// TIA Portal V17 program export: 2 tag tables, 1 data types, 3 data blocks, 33 code blocks (in call order from the OBs), 23 instance data blocks

VAR_GLOBAL   // PLC tag table "Default tag table"
   System_Byte AT %MB1 : Byte;
   FirstScan AT %M1.0 : Bool;
   DiagStatusUpdate AT %M1.1 : Bool;
   Clock_Byte AT %MB0 : Byte;
   Clock_10Hz AT %M0.0 : Bool;
   Clock_5Hz AT %M0.1 : Bool;
   "Clock_2.5Hz" AT %M0.2 : Bool;
   Clock_2Hz AT %M0.3 : Bool;
   "Clock_1.25Hz" AT %M0.4 : Bool;
   Clock_1Hz AT %M0.5 : Bool;
   "Clock_0.625Hz" AT %M0.6 : Bool;
   "Clock_0.5Hz" AT %M0.7 : Bool;
   "System_Byte(1)" AT %MB1 : Byte;
   AlwaysTRUE AT %M1.2 : Bool;
   AlwaysFALSE AT %M1.3 : Bool;
   Tag_1 AT %Q0.0 : Bool;
   Tag_2 AT %Q0.7 : Bool;
END_VAR

VAR_GLOBAL   // PLC tag table "System_Tags"
   pulse_01s AT %M10.0 : Bool;
   pulse_05s AT %M10.1 : Bool;
   pulse_1s AT %M10.2 : Bool;
   pulse_5s AT %M10.3 : Bool;
   pulse_10s AT %M10.4 : Bool;
   pulse_30s AT %M10.5 : Bool;
   pulse_1m AT %M10.6 : Bool;
   pulse_5m AT %M10.7 : Bool;
   pulse_10m AT %M11.0 : Bool;
   pulse_1h AT %M11.2 : Bool;
   TRUE AT %M1.2 : Bool;
   FALSE AT %M1.3 : Bool;
   Hand_DI AT %M12.0 : Bool;
   Hand_DO AT %M12.1 : Bool;
   Hand_AI AT %M12.2 : Bool;
   Hand_AO AT %M12.3 : Bool;
   Hand_M AT %M12.4 : Bool;
   Hand_MD AT %M12.5 : Bool;
   Hand_MDA AT %M12.6 : Bool;
   Hand_V AT %M12.7 : Bool;
   Hand_VD2 AT %M13.0 : Bool;
   Hand_VDA AT %M13.1 : Bool;
   Hand_Any AT %M13.7 : Bool;
   Alm_AI AT %M14.0 : Bool;
   Alm_M AT %M14.1 : Bool;
   Alm_MD AT %M14.2 : Bool;
   Alm_MDA AT %M14.3 : Bool;
   Alm_V AT %M14.4 : Bool;
   Alm_VD2 AT %M14.5 : Bool;
   Alm_VDA AT %M14.6 : Bool;
   Alm_Logick AT %M14.7 : Bool;
   Alm_Any AT %M15.7 : Bool;
   All_Block AT %M2.0 : Bool;
   Reset_All AT %M3.0 : Bool;
   Local_Mode AT %M4.0 : Bool;
   Sim_All AT %M5.0 : Bool;
   AI_Val_1 AT %MB100 : Byte;
   AI_Val_2 AT %MB101 : Byte;
   AI_Value AT %MW100 : Word;
   AO_Val_1 AT %MB102 : Byte;
   AO_Val_2 AT %MB103 : Byte;
   AO_Value AT %MW102 : Word;
   Events AT %MW200 : Word;
   pulse_1_day AT %M11.3 : Bool;
   pulse_1_week AT %M11.4 : Bool;
   pulse_1_month AT %M11.5 : Bool;
   pulse_30m AT %M11.1 : Bool;
   pulse_s1 AT %M11.6 : Bool;
   pulse_s2 AT %M11.7 : Bool;
   Hand_Low AT %M13.5 : Bool;
   Hand_High AT %M13.6 : Bool;
   Reset_Hand AT %M3.1 : Bool;
   Events_pos AT %MW210 : Word;
   Alarms AT %MW202 : Word;
   Alarms_pos AT %MW212 : Word;
END_VAR

TYPE "CMD"
// stored: IsFailsafeCompliant false
   STRUCT
      Start_A : Bool;   // Автозапуск / Запуск в авторежиме
      Start_M : Bool;   // Ручной - вперёд / Запуск в ручном режиме
      Hand : Bool;   // 0 - авто, 1 - ручной / 0 - Авто, 1 - Ручной
      Local : Bool;   // Локальный
      Lock : Bool;   // Блокировать / Блокировка
      Service : Bool;   // Сервис
      Safety : Bool;   // Безопасность
      Force : Bool;   // Принудительный
      Alarm : Bool;   // Есть авария / Авария
      Reset : Bool;   // Сброс аварий
      Sim : Bool;   // Режим симуляции
      Vector { S7_SetPoint := 'True'} : Bool;   // Выбор направления
      ResetOpTime : Bool;   // Сброс счётчика наработки
      Ready : Bool := true;   // Разрешение дистанционного управления
      reserv : Bool;
   END_STRUCT;
END_TYPE

DATA_BLOCK "FE_DB"   // DB5
{ S7_Optimized_Access := 'FALSE' }
VERSION : 0.1
// stored: AutoNumber false, DBAccessibleFromOPCUA true, IsOnlyStoredInLoadMemory false, IsWriteProtectedInAS false
   VAR RETAIN
      FE : Array[0..1] of Struct   // Чтение - Input Register (04), Запись - Holding Register (06)
         Flow_Out : Real;   // Накопленный объем +
         Flow_In : Real;   // Накопленный объём -
         Flow : Real;   // Мгновенный расход
         TE_1 : Real;   // Температура канала 1, С
         TE_2 : Real;   // Температура канала 2, С
         PE : Real;   // Давление среды, кПа
         Use { S7_SetPoint := 'True'} : Bool;
         Link : Bool;
         NoRead : Bool;
         NoWrite : Bool;
         ID { S7_SetPoint := 'True'} : Int;
         ADDR { S7_SetPoint := 'True'} : UInt;
         "Name" { S7_SetPoint := 'True'} : String[10];
      END_STRUCT;
   END_VAR
BEGIN
   FE[0].Use := FALSE;
   FE[1].Use := TRUE;
   FE[0].ID := 0;
   FE[1].ID := 1;
   FE[0].ADDR := 0;
   FE[1].ADDR := 41;
   FE[0]."Name" := '';
   FE[1]."Name" := 'FE';
END_DATA_BLOCK

DATA_BLOCK "tGw_DB"   // DB3
{ S7_Optimized_Access := 'TRUE' }
VERSION : 0.1
// stored: AutoNumber true, DBAccessibleFromOPCUA true, IsOnlyStoredInLoadMemory false, IsRetainMemResEnabled false, IsWriteProtectedInAS false, MemoryReserve 100
   VAR RETAIN
      tGw : Array[0..1] of Struct   // Точка подключения к КП
         IP { S7_SetPoint := 'True'} : IP_V4;
         Port { S7_SetPoint := 'True'} : UInt;
      END_STRUCT;
      "Name" { S7_SetPoint := 'True'} : WString[10] := WSTRING#'1';
      ID { S7_SetPoint := 'True'} : Int := 0;
   END_VAR
BEGIN
   tGw[0].IP.ADDR[1] := 16#0A;
   tGw[0].IP.ADDR[2..3] := 16#01;
   tGw[0].IP.ADDR[4] := 16#9B;
   tGw[1].IP.ADDR[1] := 16#0A;
   tGw[1].IP.ADDR[2..3] := 16#01;
   tGw[1].IP.ADDR[4] := 16#C9;
   tGw[0..1].Port := 503;
END_DATA_BLOCK

DATA_BLOCK "Support_DB"   // DB1000
{ S7_Optimized_Access := 'TRUE' }
VERSION : 0.1
// stored: AutoNumber false, DBAccessibleFromOPCUA true, IsOnlyStoredInLoadMemory false, IsRetainMemResEnabled false, IsWriteProtectedInAS false, MemoryReserve 100
   VAR
      DTR_Clean : Bool;   // Очистка DTR
      DTR_1 : Int;   // Data Transfer 1
      DTR_2 : Int;   // Data Transfer 2
      DTR_3 : Int;   // Data Transfer 3
   END_VAR
   VAR RETAIN
      All_AIs { S7_SetPoint := 'True'} : Int := 399;   // Номер последнего DB аналоговых входов
      All_AOs { S7_SetPoint := 'True'} : Int := 499;   // Номер последнего DB аналоговых выходов
      All_DIs { S7_SetPoint := 'True'} : Int := 209;   // Номер последнего DB дискретных входов
      All_DOs { S7_SetPoint := 'True'} : Int := 219;   // Номер последнего DB дискретных выходов
      All_MDs { S7_SetPoint := 'True'} : Int := 599;   // Номер последнего DB двигателей без ЧП
      All_MDAs { S7_SetPoint := 'True'} : Int := 699;   // Номер последнего DB двигателей с ЧП
      All_VD2s { S7_SetPoint := 'True'} : Int := 799;   // Номер последнего DB заслонки
      All_VD2As { S7_SetPoint := 'True'} : Int := 899;   // Номер последнего DB заслонки с позиционированием
      All_PIDs { S7_SetPoint := 'True'} : Int := 999;   // Номер последнего DB для PID-регулятора
   END_VAR
BEGIN
END_DATA_BLOCK

ORGANIZATION_BLOCK "Main"   // OB1, LAD, ProgramCycle
TITLE = "Main Program Sweep (Cycle)"
{ S7_Optimized_Access := 'TRUE' }
VERSION : 0.1
// stored: AutoNumber true, IsIECCheckEnabled false, SetENOAutomatically false
   VAR_INPUT
      Initial_Call : Bool;   // Initial call of this OB
      Remanence : Bool;   // =True, if remanent data are available
   END_VAR
   VAR_TEMP   // added for the SCL form of the ladder/FBD networks
      _w1 : Bool;
   END_VAR
BEGIN

REGION Network 1
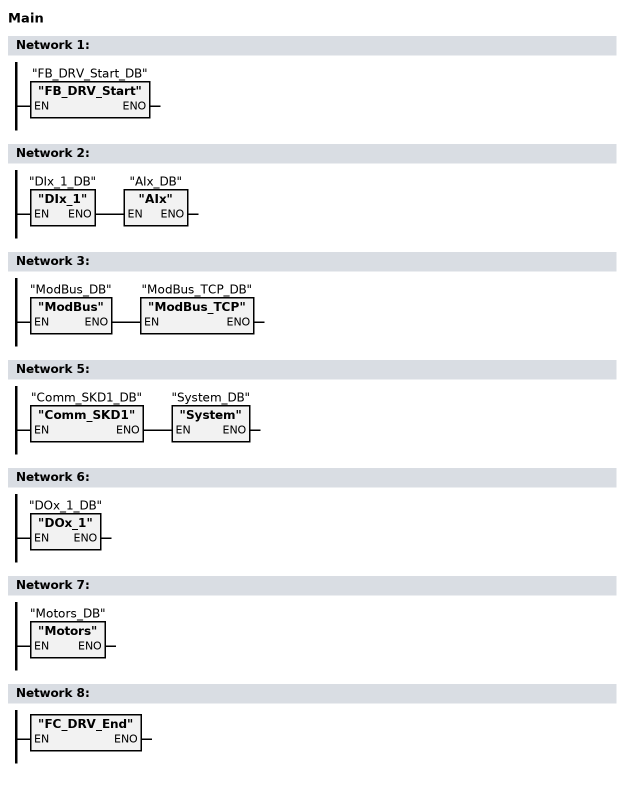
   RUNG wire#powerrail
      "FB_DRV_Start_DB"()
   END_RUNG
   // the same network as SCL:
   "FB_DRV_Start_DB"();   // "FB_DRV_Start"
END_REGION

REGION Network 2
   RUNG wire#powerrail
      "DIx_1_DB"()
      "AIx_DB"()
   END_RUNG
   // the same network as SCL:
   "DIx_1_DB"(ENO => #_w1);   // "DIx_1"
   IF #_w1 THEN
       "AIx_DB"();   // "AIx"
   END_IF;
END_REGION

REGION Network 3
   RUNG wire#powerrail
      "ModBus_DB"()
      "ModBus_TCP_DB"()
   END_RUNG
   // the same network as SCL:
   "ModBus_DB"(ENO => #_w1);   // "ModBus"
   IF #_w1 THEN
       "ModBus_TCP_DB"();   // "ModBus_TCP"
   END_IF;
END_REGION

REGION Network 5
   RUNG wire#powerrail
      "Comm_SKD1_DB"()
      "System_DB"()
   END_RUNG
   // the same network as SCL:
   "Comm_SKD1_DB"(ENO => #_w1);   // "Comm_SKD1"
   IF #_w1 THEN
       "System_DB"();   // "System"
   END_IF;
END_REGION

REGION Network 6
   RUNG wire#powerrail
      "DOx_1_DB"()
   END_RUNG
   // the same network as SCL:
   "DOx_1_DB"();   // "DOx_1"
END_REGION

REGION Network 7
   RUNG wire#powerrail
      "Motors_DB"()
   END_RUNG
   // the same network as SCL:
   "Motors_DB"();   // "Motors"
END_REGION

REGION Network 8
   RUNG wire#powerrail
      "FC_DRV_End"()
   END_RUNG
   // the same network as SCL:
   "FC_DRV_End"();
END_REGION
END_ORGANIZATION_BLOCK

FUNCTION_BLOCK "FB_DRV_Start"   // FB100, LAD
{ S7_Optimized_Access := 'TRUE' }
VERSION : 0.1
// stored: AutoNumber false, IsIECCheckEnabled false, IsRetainMemResEnabled false, MemoryReserve 100, SetENOAutomatically false, UDAEnableTagReadback false
   VAR
      last_01s : Int;
      last_05s : Int;
      last_1s : Int;
      last_5s : Int;
      last_10s : Int;
      last_30s : Int;
      last_1m : Int;
      last_5m : Int;
      last_10m : Int;
      last_30m : Int;
      last_1h : Int;
      last_1_day : Int;
      last_1_week : Int;
      last_1_month : Int;
      last_s1 : Int;
      last_s2 : Int;
      "1h_minutes" { S7_SetPoint := 'True'} : Int;
      "1_day_hour" { S7_SetPoint := 'True'} : Int;
      "1_day_minutes" { S7_SetPoint := 'True'} : Int;
      "1_week_weekday" { S7_SetPoint := 'True'} : Int := 1;
      "1_week_hour" { S7_SetPoint := 'True'} : Int;
      "1_week_minutes" { S7_SetPoint := 'True'} : Int;
      "1_month_date" { S7_SetPoint := 'True'} : Int := 1;
      "1_month_hour" { S7_SetPoint := 'True'} : Int;
      "1_month_minutes" { S7_SetPoint := 'True'} : Int;
      s1_hour : Int := 8;
      s1_minutes : Int;
      s2_hour : Int := 20;
      s2_minutes : Int;
      pos : Array[0..15] of Bool;
      Error : Word;
   END_VAR
   VAR_TEMP
      cnt_01s : Int;
      cnt_5s : Int;
      cnt_10s : Int;
      cnt_30s : Int;
      cnt_5m : Int;
      cnt_10m : Int;
      cnt_30m : Int;
   END_VAR
   VAR_TEMP   // added for the SCL form of the ladder/FBD networks
      _w1 : Bool;
      _w2 : Bool;
   END_VAR
BEGIN

REGION Network 1: Обработчик системного времени
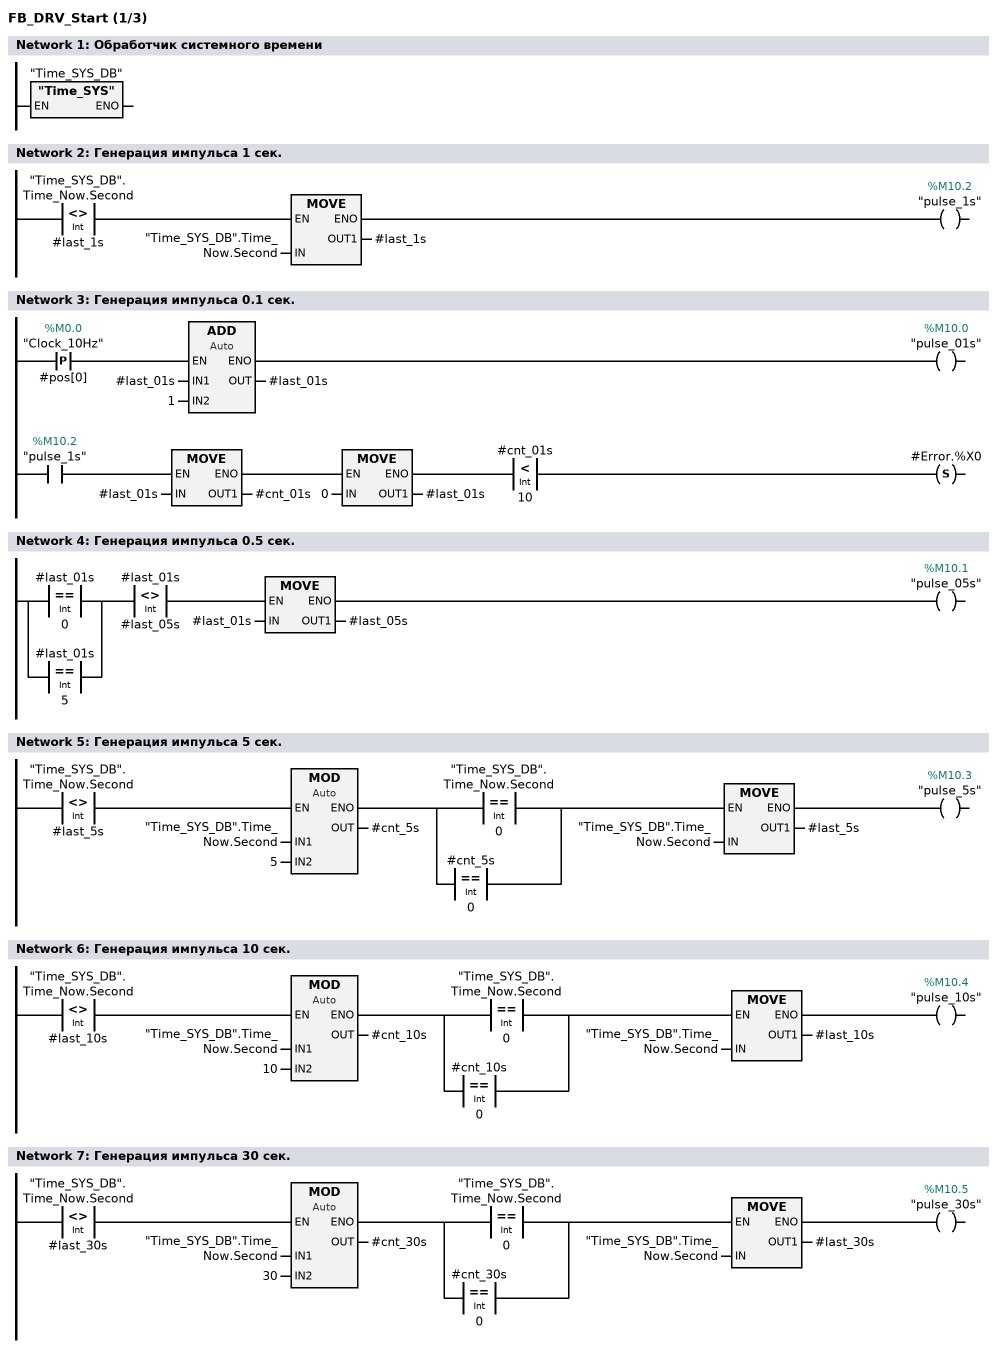
   RUNG wire#powerrail
      "Time_SYS_DB"()
   END_RUNG
   // the same network as SCL:
   "Time_SYS_DB"();   // "Time_SYS"
END_REGION

REGION Network 2: Генерация импульса 1 сек.
   RUNG wire#powerrail
      { S7_Templates := "SrcType := Int" } NE_Contact(in1 := "Time_SYS_DB".Time_Now.Second, in2 := #last_1s)
      Move(in := "Time_SYS_DB".Time_Now.Second, out1 => #last_1s)
      Coil( "pulse_1s" )
   END_RUNG
   // the same network as SCL:
   #_w1 := "Time_SYS_DB".Time_Now.Second <> #last_1s;
   IF #_w1 THEN #last_1s := "Time_SYS_DB".Time_Now.Second; END_IF;
   "pulse_1s" := #_w1;
END_REGION

REGION Network 3: Генерация импульса 0.1 сек.
   RUNG wire#powerrail
      P_Contact(operand := "Clock_10Hz", bit := #pos[0])
      Add(in1 := #last_01s, in2 := 1, out => #last_01s)
      Coil( "pulse_01s" )
   END_RUNG
   RUNG wire#powerrail
      Contact( "pulse_1s" )
      Move(in := #last_01s, out1 => #cnt_01s)
      Move(in := 0, out1 => #last_01s)
      { S7_Templates := "SrcType := Int" } LT_Contact(in1 := #cnt_01s, in2 := 10)
      S_Coil( #Error.%X0 )
   END_RUNG
   // the same network as SCL:
   #_w1 := "Clock_10Hz" AND NOT #pos[0];   // rising edge of "Clock_10Hz"
   #pos[0] := "Clock_10Hz";
   IF #_w1 THEN #last_01s := #last_01s + 1; END_IF;
   "pulse_01s" := #_w1;
   IF "pulse_1s" THEN
       #cnt_01s := #last_01s;
       #last_01s := 0;
   END_IF;
   IF "pulse_1s" AND (#cnt_01s < 10) THEN #Error.%X0 := TRUE; END_IF;
END_REGION

REGION Network 4: Генерация импульса 0.5 сек.
   RUNG wire#powerrail
      { S7_Templates := "SrcType := Int" } EQ_Contact(in1 := #last_01s, in2 := 0)
      wire#w1
      { S7_Templates := "SrcType := Int" } NE_Contact(in1 := #last_01s, in2 := #last_05s)
      Move(in := #last_01s, out1 => #last_05s)
      Coil( "pulse_05s" )
   END_RUNG
   RUNG wire#powerrail
      { S7_Templates := "SrcType := Int" } EQ_Contact(in1 := #last_01s, in2 := 5)
   END_RUNG wire#w1
   // the same network as SCL:
   #_w1 := ((#last_01s = 0) OR (#last_01s = 5)) AND (#last_01s <> #last_05s);
   IF #_w1 THEN #last_05s := #last_01s; END_IF;
   "pulse_05s" := #_w1;
END_REGION

REGION Network 5: Генерация импульса 5 сек.
   RUNG wire#powerrail
      { S7_Templates := "SrcType := Int" } NE_Contact(in1 := "Time_SYS_DB".Time_Now.Second, in2 := #last_5s)
      Mod(in1 := "Time_SYS_DB".Time_Now.Second, in2 := 5, out => #cnt_5s)
      wire#w1
      { S7_Templates := "SrcType := Int" } EQ_Contact(in1 := "Time_SYS_DB".Time_Now.Second, in2 := 0)
      wire#w2
      Move(in := "Time_SYS_DB".Time_Now.Second, out1 => #last_5s)
      Coil( "pulse_5s" )
   END_RUNG
   RUNG wire#w1
      { S7_Templates := "SrcType := Int" } EQ_Contact(in1 := #cnt_5s, in2 := 0)
   END_RUNG wire#w2
   // the same network as SCL:
   #_w1 := "Time_SYS_DB".Time_Now.Second <> #last_5s;
   IF #_w1 THEN #cnt_5s := "Time_SYS_DB".Time_Now.Second MOD 5; END_IF;
   #_w2 := #_w1 AND (("Time_SYS_DB".Time_Now.Second = 0) OR (#cnt_5s = 0));
   IF #_w2 THEN #last_5s := "Time_SYS_DB".Time_Now.Second; END_IF;
   "pulse_5s" := #_w2;
END_REGION

REGION Network 6: Генерация импульса 10 сек.
   RUNG wire#powerrail
      { S7_Templates := "SrcType := Int" } NE_Contact(in1 := "Time_SYS_DB".Time_Now.Second, in2 := #last_10s)
      Mod(in1 := "Time_SYS_DB".Time_Now.Second, in2 := 10, out => #cnt_10s)
      wire#w1
      { S7_Templates := "SrcType := Int" } EQ_Contact(in1 := "Time_SYS_DB".Time_Now.Second, in2 := 0)
      wire#w2
      Move(in := "Time_SYS_DB".Time_Now.Second, out1 => #last_10s)
      Coil( "pulse_10s" )
   END_RUNG
   RUNG wire#w1
      { S7_Templates := "SrcType := Int" } EQ_Contact(in1 := #cnt_10s, in2 := 0)
   END_RUNG wire#w2
   // the same network as SCL:
   #_w1 := "Time_SYS_DB".Time_Now.Second <> #last_10s;
   IF #_w1 THEN #cnt_10s := "Time_SYS_DB".Time_Now.Second MOD 10; END_IF;
   #_w2 := #_w1 AND (("Time_SYS_DB".Time_Now.Second = 0) OR (#cnt_10s = 0));
   IF #_w2 THEN #last_10s := "Time_SYS_DB".Time_Now.Second; END_IF;
   "pulse_10s" := #_w2;
END_REGION

REGION Network 7: Генерация импульса 30 сек.
   RUNG wire#powerrail
      { S7_Templates := "SrcType := Int" } NE_Contact(in1 := "Time_SYS_DB".Time_Now.Second, in2 := #last_30s)
      Mod(in1 := "Time_SYS_DB".Time_Now.Second, in2 := 30, out => #cnt_30s)
      wire#w1
      { S7_Templates := "SrcType := Int" } EQ_Contact(in1 := "Time_SYS_DB".Time_Now.Second, in2 := 0)
      wire#w2
      Move(in := "Time_SYS_DB".Time_Now.Second, out1 => #last_30s)
      Coil( "pulse_30s" )
   END_RUNG
   RUNG wire#w1
      { S7_Templates := "SrcType := Int" } EQ_Contact(in1 := #cnt_30s, in2 := 0)
   END_RUNG wire#w2
   // the same network as SCL:
   #_w1 := "Time_SYS_DB".Time_Now.Second <> #last_30s;
   IF #_w1 THEN #cnt_30s := "Time_SYS_DB".Time_Now.Second MOD 30; END_IF;
   #_w2 := #_w1 AND (("Time_SYS_DB".Time_Now.Second = 0) OR (#cnt_30s = 0));
   IF #_w2 THEN #last_30s := "Time_SYS_DB".Time_Now.Second; END_IF;
   "pulse_30s" := #_w2;
END_REGION

REGION Network 8: Генерация импульса 1 мин.
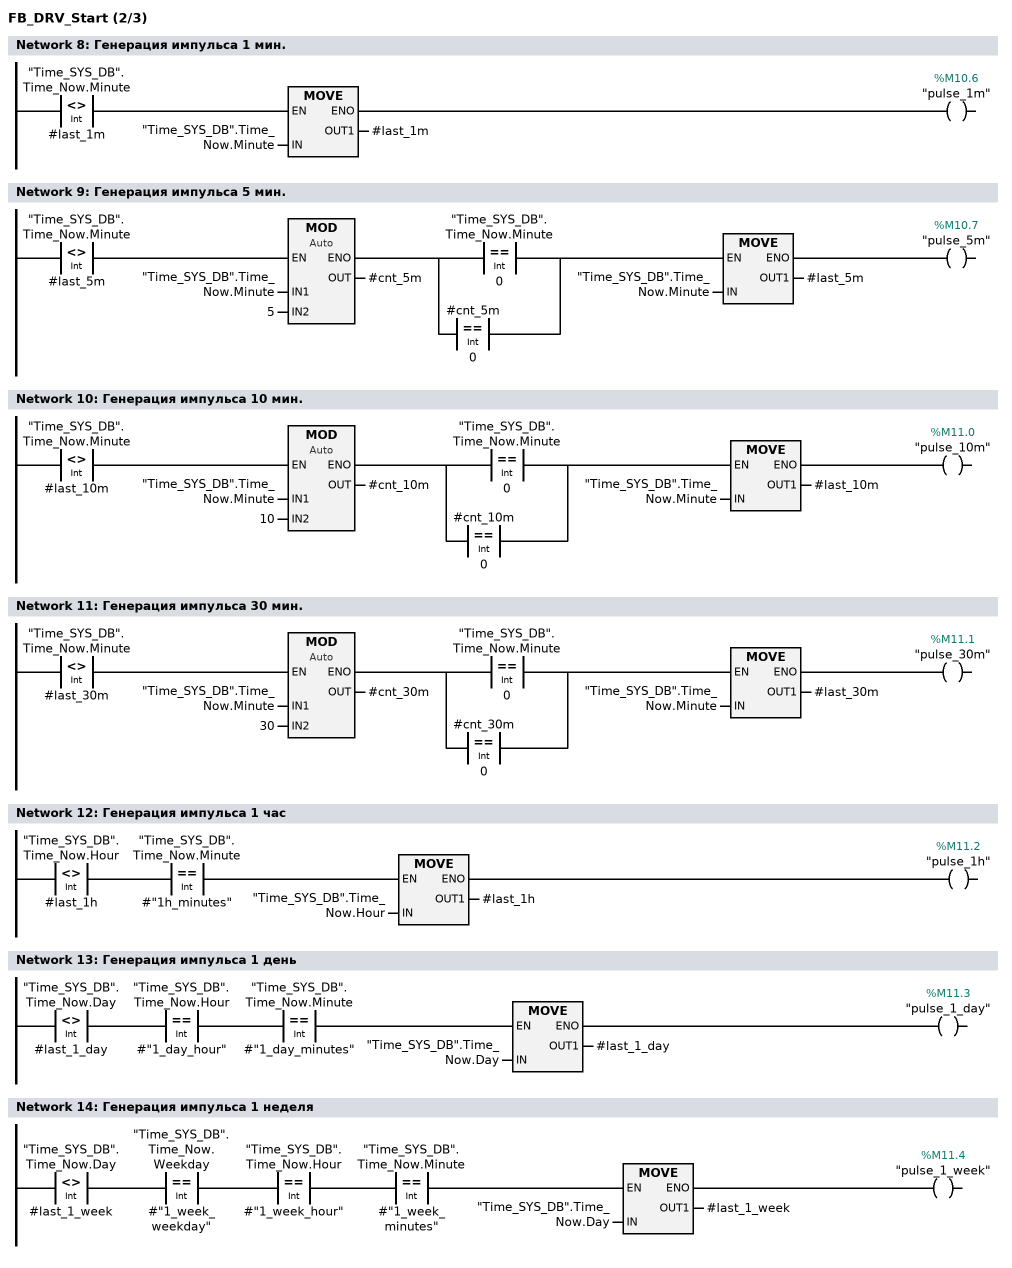
   RUNG wire#powerrail
      { S7_Templates := "SrcType := Int" } NE_Contact(in1 := "Time_SYS_DB".Time_Now.Minute, in2 := #last_1m)
      Move(in := "Time_SYS_DB".Time_Now.Minute, out1 => #last_1m)
      Coil( "pulse_1m" )
   END_RUNG
   // the same network as SCL:
   #_w1 := "Time_SYS_DB".Time_Now.Minute <> #last_1m;
   IF #_w1 THEN #last_1m := "Time_SYS_DB".Time_Now.Minute; END_IF;
   "pulse_1m" := #_w1;
END_REGION

REGION Network 9: Генерация импульса 5 мин.
   RUNG wire#powerrail
      { S7_Templates := "SrcType := Int" } NE_Contact(in1 := "Time_SYS_DB".Time_Now.Minute, in2 := #last_5m)
      Mod(in1 := "Time_SYS_DB".Time_Now.Minute, in2 := 5, out => #cnt_5m)
      wire#w1
      { S7_Templates := "SrcType := Int" } EQ_Contact(in1 := "Time_SYS_DB".Time_Now.Minute, in2 := 0)
      wire#w2
      Move(in := "Time_SYS_DB".Time_Now.Minute, out1 => #last_5m)
      Coil( "pulse_5m" )
   END_RUNG
   RUNG wire#w1
      { S7_Templates := "SrcType := Int" } EQ_Contact(in1 := #cnt_5m, in2 := 0)
   END_RUNG wire#w2
   // the same network as SCL:
   #_w1 := "Time_SYS_DB".Time_Now.Minute <> #last_5m;
   IF #_w1 THEN #cnt_5m := "Time_SYS_DB".Time_Now.Minute MOD 5; END_IF;
   #_w2 := #_w1 AND (("Time_SYS_DB".Time_Now.Minute = 0) OR (#cnt_5m = 0));
   IF #_w2 THEN #last_5m := "Time_SYS_DB".Time_Now.Minute; END_IF;
   "pulse_5m" := #_w2;
END_REGION

REGION Network 10: Генерация импульса 10 мин.
   RUNG wire#powerrail
      { S7_Templates := "SrcType := Int" } NE_Contact(in1 := "Time_SYS_DB".Time_Now.Minute, in2 := #last_10m)
      Mod(in1 := "Time_SYS_DB".Time_Now.Minute, in2 := 10, out => #cnt_10m)
      wire#w1
      { S7_Templates := "SrcType := Int" } EQ_Contact(in1 := "Time_SYS_DB".Time_Now.Minute, in2 := 0)
      wire#w2
      Move(in := "Time_SYS_DB".Time_Now.Minute, out1 => #last_10m)
      Coil( "pulse_10m" )
   END_RUNG
   RUNG wire#w1
      { S7_Templates := "SrcType := Int" } EQ_Contact(in1 := #cnt_10m, in2 := 0)
   END_RUNG wire#w2
   // the same network as SCL:
   #_w1 := "Time_SYS_DB".Time_Now.Minute <> #last_10m;
   IF #_w1 THEN #cnt_10m := "Time_SYS_DB".Time_Now.Minute MOD 10; END_IF;
   #_w2 := #_w1 AND (("Time_SYS_DB".Time_Now.Minute = 0) OR (#cnt_10m = 0));
   IF #_w2 THEN #last_10m := "Time_SYS_DB".Time_Now.Minute; END_IF;
   "pulse_10m" := #_w2;
END_REGION

REGION Network 11: Генерация импульса 30 мин.
   RUNG wire#powerrail
      { S7_Templates := "SrcType := Int" } NE_Contact(in1 := "Time_SYS_DB".Time_Now.Minute, in2 := #last_30m)
      Mod(in1 := "Time_SYS_DB".Time_Now.Minute, in2 := 30, out => #cnt_30m)
      wire#w1
      { S7_Templates := "SrcType := Int" } EQ_Contact(in1 := "Time_SYS_DB".Time_Now.Minute, in2 := 0)
      wire#w2
      Move(in := "Time_SYS_DB".Time_Now.Minute, out1 => #last_30m)
      Coil( "pulse_30m" )
   END_RUNG
   RUNG wire#w1
      { S7_Templates := "SrcType := Int" } EQ_Contact(in1 := #cnt_30m, in2 := 0)
   END_RUNG wire#w2
   // the same network as SCL:
   #_w1 := "Time_SYS_DB".Time_Now.Minute <> #last_30m;
   IF #_w1 THEN #cnt_30m := "Time_SYS_DB".Time_Now.Minute MOD 30; END_IF;
   #_w2 := #_w1 AND (("Time_SYS_DB".Time_Now.Minute = 0) OR (#cnt_30m = 0));
   IF #_w2 THEN #last_30m := "Time_SYS_DB".Time_Now.Minute; END_IF;
   "pulse_30m" := #_w2;
END_REGION

REGION Network 12: Генерация импульса 1 час
   RUNG wire#powerrail
      { S7_Templates := "SrcType := Int" } NE_Contact(in1 := "Time_SYS_DB".Time_Now.Hour, in2 := #last_1h)
      { S7_Templates := "SrcType := Int" } EQ_Contact(in1 := "Time_SYS_DB".Time_Now.Minute, in2 := #"1h_minutes")
      Move(in := "Time_SYS_DB".Time_Now.Hour, out1 => #last_1h)
      Coil( "pulse_1h" )
   END_RUNG
   // the same network as SCL:
   #_w1 := ("Time_SYS_DB".Time_Now.Hour <> #last_1h) AND ("Time_SYS_DB".Time_Now.Minute = #"1h_minutes");
   IF #_w1 THEN #last_1h := "Time_SYS_DB".Time_Now.Hour; END_IF;
   "pulse_1h" := #_w1;
END_REGION

REGION Network 13: Генерация импульса 1 день
   RUNG wire#powerrail
      { S7_Templates := "SrcType := Int" } NE_Contact(in1 := "Time_SYS_DB".Time_Now.Day, in2 := #last_1_day)
      { S7_Templates := "SrcType := Int" } EQ_Contact(in1 := "Time_SYS_DB".Time_Now.Hour, in2 := #"1_day_hour")
      { S7_Templates := "SrcType := Int" } EQ_Contact(in1 := "Time_SYS_DB".Time_Now.Minute, in2 := #"1_day_minutes")
      Move(in := "Time_SYS_DB".Time_Now.Day, out1 => #last_1_day)
      Coil( "pulse_1_day" )
   END_RUNG
   // the same network as SCL:
   #_w1 := ("Time_SYS_DB".Time_Now.Day <> #last_1_day) AND ("Time_SYS_DB".Time_Now.Hour = #"1_day_hour") AND ("Time_SYS_DB".Time_Now.Minute = #"1_day_minutes");
   IF #_w1 THEN #last_1_day := "Time_SYS_DB".Time_Now.Day; END_IF;
   "pulse_1_day" := #_w1;
END_REGION

REGION Network 14: Генерация импульса 1 неделя
   RUNG wire#powerrail
      { S7_Templates := "SrcType := Int" } NE_Contact(in1 := "Time_SYS_DB".Time_Now.Day, in2 := #last_1_week)
      { S7_Templates := "SrcType := Int" } EQ_Contact(in1 := "Time_SYS_DB".Time_Now.Weekday, in2 := #"1_week_weekday")
      { S7_Templates := "SrcType := Int" } EQ_Contact(in1 := "Time_SYS_DB".Time_Now.Hour, in2 := #"1_week_hour")
      { S7_Templates := "SrcType := Int" } EQ_Contact(in1 := "Time_SYS_DB".Time_Now.Minute, in2 := #"1_week_minutes")
      Move(in := "Time_SYS_DB".Time_Now.Day, out1 => #last_1_week)
      Coil( "pulse_1_week" )
   END_RUNG
   // the same network as SCL:
   #_w1 := ("Time_SYS_DB".Time_Now.Day <> #last_1_week) AND ("Time_SYS_DB".Time_Now.Weekday = #"1_week_weekday") AND ("Time_SYS_DB".Time_Now.Hour = #"1_week_hour") AND ("Time_SYS_DB".Time_Now.Minute = #"1_week_minutes");
   IF #_w1 THEN #last_1_week := "Time_SYS_DB".Time_Now.Day; END_IF;
   "pulse_1_week" := #_w1;
END_REGION

REGION Network 15: Генерация импульса 1 месяц
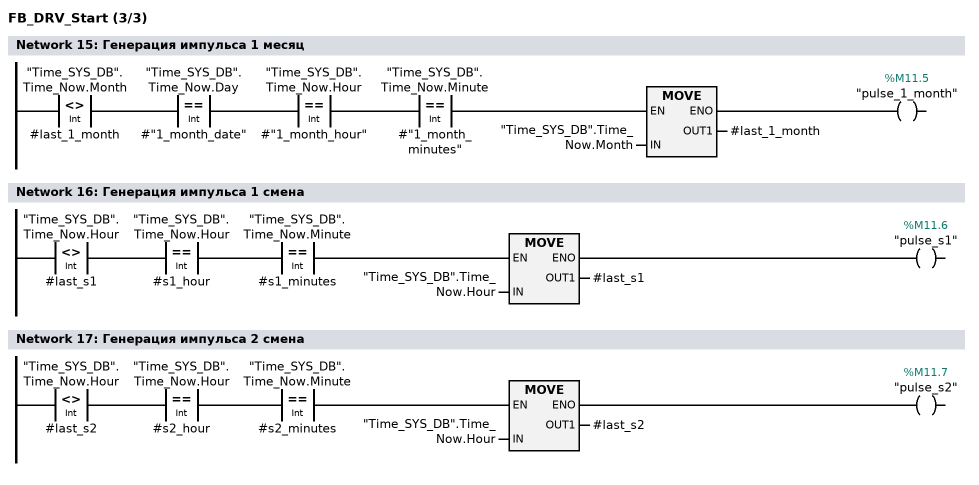
   RUNG wire#powerrail
      { S7_Templates := "SrcType := Int" } NE_Contact(in1 := "Time_SYS_DB".Time_Now.Month, in2 := #last_1_month)
      { S7_Templates := "SrcType := Int" } EQ_Contact(in1 := "Time_SYS_DB".Time_Now.Day, in2 := #"1_month_date")
      { S7_Templates := "SrcType := Int" } EQ_Contact(in1 := "Time_SYS_DB".Time_Now.Hour, in2 := #"1_month_hour")
      { S7_Templates := "SrcType := Int" } EQ_Contact(in1 := "Time_SYS_DB".Time_Now.Minute, in2 := #"1_month_minutes")
      Move(in := "Time_SYS_DB".Time_Now.Month, out1 => #last_1_month)
      Coil( "pulse_1_month" )
   END_RUNG
   // the same network as SCL:
   #_w1 := ("Time_SYS_DB".Time_Now.Month <> #last_1_month) AND ("Time_SYS_DB".Time_Now.Day = #"1_month_date") AND ("Time_SYS_DB".Time_Now.Hour = #"1_month_hour") AND ("Time_SYS_DB".Time_Now.Minute = #"1_month_minutes");
   IF #_w1 THEN #last_1_month := "Time_SYS_DB".Time_Now.Month; END_IF;
   "pulse_1_month" := #_w1;
END_REGION

REGION Network 16: Генерация импульса 1 смена
   RUNG wire#powerrail
      { S7_Templates := "SrcType := Int" } NE_Contact(in1 := "Time_SYS_DB".Time_Now.Hour, in2 := #last_s1)
      { S7_Templates := "SrcType := Int" } EQ_Contact(in1 := "Time_SYS_DB".Time_Now.Hour, in2 := #s1_hour)
      { S7_Templates := "SrcType := Int" } EQ_Contact(in1 := "Time_SYS_DB".Time_Now.Minute, in2 := #s1_minutes)
      Move(in := "Time_SYS_DB".Time_Now.Hour, out1 => #last_s1)
      Coil( "pulse_s1" )
   END_RUNG
   // the same network as SCL:
   #_w1 := ("Time_SYS_DB".Time_Now.Hour <> #last_s1) AND ("Time_SYS_DB".Time_Now.Hour = #s1_hour) AND ("Time_SYS_DB".Time_Now.Minute = #s1_minutes);
   IF #_w1 THEN #last_s1 := "Time_SYS_DB".Time_Now.Hour; END_IF;
   "pulse_s1" := #_w1;
END_REGION

REGION Network 17: Генерация импульса 2 смена
   RUNG wire#powerrail
      { S7_Templates := "SrcType := Int" } NE_Contact(in1 := "Time_SYS_DB".Time_Now.Hour, in2 := #last_s2)
      { S7_Templates := "SrcType := Int" } EQ_Contact(in1 := "Time_SYS_DB".Time_Now.Hour, in2 := #s2_hour)
      { S7_Templates := "SrcType := Int" } EQ_Contact(in1 := "Time_SYS_DB".Time_Now.Minute, in2 := #s2_minutes)
      Move(in := "Time_SYS_DB".Time_Now.Hour, out1 => #last_s2)
      Coil( "pulse_s2" )
   END_RUNG
   // the same network as SCL:
   #_w1 := ("Time_SYS_DB".Time_Now.Hour <> #last_s2) AND ("Time_SYS_DB".Time_Now.Hour = #s2_hour) AND ("Time_SYS_DB".Time_Now.Minute = #s2_minutes);
   IF #_w1 THEN #last_s2 := "Time_SYS_DB".Time_Now.Hour; END_IF;
   "pulse_s2" := #_w1;
END_REGION
END_FUNCTION_BLOCK

FUNCTION_BLOCK "Time_SYS"   // FB95, LAD
{ S7_Optimized_Access := 'FALSE' }
VERSION : 0.1
// stored: AutoNumber false, IsIECCheckEnabled false, SetENOAutomatically false, UDAEnableTagReadback false
   VAR DB_SPECIFIC
      Set_Time : Bool;   // Заданное время
      Time_Now : Struct   // Текущее время
         Year : Int;   // год
         Month : Int;   // месяц
         Day : Int;   // день месяца
         Weekday : Int;   // день недели (1 - воскресенье)
         Hour : Int;   // часы
         Minute : Int;   // минуты
         Second : Int;   // секунды
      END_STRUCT;
      Time_SP : Struct   // Текущее время
         Year : Int;   // год
         Month : Int;   // месяц
         Day : Int;   // день месяца
         Weekday : Int;   // день недели (1 - воскресенье)
         Hour : Int;   // часы
         Minute : Int;   // минуты
         Second : Int;   // секунды
      END_STRUCT;
      TimeZone { S7_SetPoint := 'True'} : TimeTransformationRule;   // Часовой пояс
      RD_SYS_Status : Int;   // Статус чтения времени
      WR_SYS_Status : Int;   // Статус записи времени
      RD_Time : DTL;   // Прочитанное сист. время
      SP_Time : DTL;   // Новое сист. время
   END_VAR
   VAR
      SET_TIMEZONE { S7_SetPoint := 'True'} : SET_TIMEZONE;   // Запись часового пояса
   END_VAR
   VAR DB_SPECIFIC
      Time_DTL : DTL;
   END_VAR
   // TimeZone.Bias := 180;   // Часовой пояс по GMT (смещение в минутах)
   // TimeZone.DaylightBias := 60;
   // TimeZone.DaylightStartMonth := 3;
   // TimeZone.DaylightStartWeek := 5;
   // TimeZone.DaylightStartWeekday := 7;
   // TimeZone.DaylightStartHour := 2;
   // TimeZone.DaylightStartMinute := 0;
   // TimeZone.StandardStartMonth := 10;
   // TimeZone.StandardStartWeek := 5;
   // TimeZone.StandardStartWeekday := 1;
   // TimeZone.StandardStartHour := 3;
   // TimeZone.StandardStartMinute := 0;
   // TimeZone.TimeZoneName := 'GMT+3';
   VAR_TEMP   // added for the SCL form of the ladder/FBD networks
      _w1 : Bool;
   END_VAR
BEGIN

REGION Network 1: Чтение системного времени
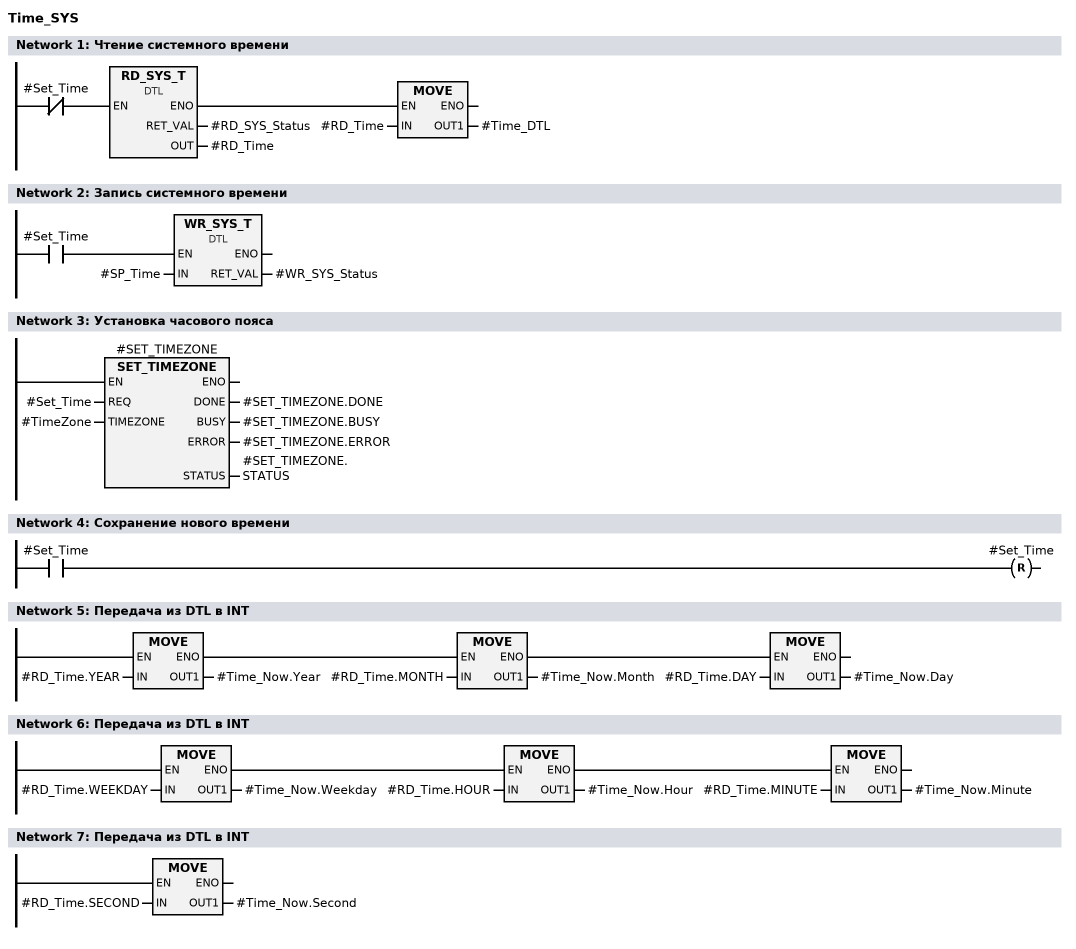
   RUNG wire#powerrail
      I_Contact( #Set_Time )
      { S7_Templates := "date_type := DTL" } RD_SYS_T(RET_VAL => #RD_SYS_Status, OUT => #RD_Time)
      Move(in := #RD_Time, out1 => #Time_DTL)
   END_RUNG
   // the same network as SCL:
   #RD_SYS_Status := RD_SYS_T(EN := NOT #Set_Time, OUT => #RD_Time, ENO => #_w1);
   IF #_w1 THEN #Time_DTL := #RD_Time; END_IF;
END_REGION

REGION Network 2: Запись системного времени
   RUNG wire#powerrail
      Contact( #Set_Time )
      { S7_Templates := "date_type := DTL" } WR_SYS_T(IN := #SP_Time, RET_VAL => #WR_SYS_Status)
   END_RUNG
   // the same network as SCL:
   IF #Set_Time THEN #WR_SYS_Status := WR_SYS_T(IN := #SP_Time); END_IF;
END_REGION

REGION Network 3: Установка часового пояса
   RUNG wire#powerrail
      #SET_TIMEZONE.SET_TIMEZONE(REQ := #Set_Time, TimeZone := #TimeZone, DONE => #SET_TIMEZONE.DONE, BUSY => #SET_TIMEZONE.BUSY, ERROR => #SET_TIMEZONE.ERROR, STATUS => #SET_TIMEZONE.STATUS)
   END_RUNG
   // the same network as SCL:
   #SET_TIMEZONE(REQ := #Set_Time,   // SET_TIMEZONE
                 TimeZone := #TimeZone,
                 DONE => #SET_TIMEZONE.DONE,
                 BUSY => #SET_TIMEZONE.BUSY,
                 ERROR => #SET_TIMEZONE.ERROR,
                 STATUS => #SET_TIMEZONE.STATUS);
END_REGION

REGION Network 4: Сохранение нового времени
   RUNG wire#powerrail
      Contact( #Set_Time )
      R_Coil( #Set_Time )
   END_RUNG
   // the same network as SCL:
   IF #Set_Time THEN #Set_Time := FALSE; END_IF;
END_REGION

REGION Network 5: Передача из DTL в INT
   RUNG wire#powerrail
      Move(in := #RD_Time.YEAR, out1 => #Time_Now.Year)
      Move(in := #RD_Time.MONTH, out1 => #Time_Now.Month)
      Move(in := #RD_Time.DAY, out1 => #Time_Now.Day)
   END_RUNG
   // the same network as SCL:
   #Time_Now.Year := #RD_Time.YEAR;
   #Time_Now.Month := #RD_Time.MONTH;
   #Time_Now.Day := #RD_Time.DAY;
END_REGION

REGION Network 6: Передача из DTL в INT
   RUNG wire#powerrail
      Move(in := #RD_Time.WEEKDAY, out1 => #Time_Now.Weekday)
      Move(in := #RD_Time.HOUR, out1 => #Time_Now.Hour)
      Move(in := #RD_Time.MINUTE, out1 => #Time_Now.Minute)
   END_RUNG
   // the same network as SCL:
   #Time_Now.Weekday := #RD_Time.WEEKDAY;
   #Time_Now.Hour := #RD_Time.HOUR;
   #Time_Now.Minute := #RD_Time.MINUTE;
END_REGION

REGION Network 7: Передача из DTL в INT
   RUNG wire#powerrail
      Move(in := #RD_Time.SECOND, out1 => #Time_Now.Second)
   END_RUNG
   // the same network as SCL:
   #Time_Now.Second := #RD_Time.SECOND;
END_REGION
END_FUNCTION_BLOCK

FUNCTION_BLOCK "DIx_1"   // FB200, LAD
{ S7_Optimized_Access := 'FALSE' }
VERSION : 0.1
// Input - входной сигнал контроллера
// pulse - частота фильтрации дребезга
// Signal - обработанный и отфильтрованный сигнал, используемый в дальнейшем
// stored: AutoNumber false, IsIECCheckEnabled false, SetENOAutomatically false, UDAEnableTagReadback false
   VAR
      AllBlock { S7_SetPoint := 'True'} : "DI_ex";   // Аварийный останов / 2.4 разрешение на работу
      "3FOk" { S7_SetPoint := 'True'} : "DI_ex";   // Питание в норме / 2.3 Нижний уровень
      Pump_Alarm { S7_SetPoint := 'True'} : "DI_ex";   // Авария насоса / Ротаметр 1
      Leak_KP { S7_SetPoint := 'True'} : "DI_ex";   // Затопление камеры КП2.7 / Ротаметр 2
      Level_Norm { S7_SetPoint := 'True'} : "DI_ex";   // Уровень в норме / Ротаметр 3
      "3Fok_1" { S7_SetPoint := 'True'} : "DI_ex";   // 3ф. сети Ввод 1 в норме / Датчик переливва
      "3Fok_2" { S7_SetPoint := 'True'} : "DI_ex";   // 3ф. сети Ввод 2 в норме / Датчик переливва
      "3Fok_sh" { S7_SetPoint := 'True'} : "DI_ex";   // 3ф. сети Ввод Шин в норме
      SHUSKV_Ok { S7_SetPoint := 'True'} : "DI_ex";   // Выключатель UC. Питание ШУСКВ в норме
      Leak_KP_res { S7_SetPoint := 'True'} : "DI_ex";
      Leak_KP_res_1 { S7_SetPoint := 'True'} : "DI_ex";
      signal_12 { S7_SetPoint := 'True'} : "DI_ex";
   END_VAR
   VAR DB_SPECIFIC
      Time_DTL { S7_SetPoint := 'True'} : DTL;
   END_VAR
   // AllBlock.ADDR_Bit := 3;
   // "3FOk".ADDR_Bit := 0;
   // Pump_Alarm.ADDR_Bit := 2;
   // Leak_KP.ADDR_Bit := 4;
   // Level_Norm.ADDR_Bit := 5;
   // "3Fok_1".ADDR_Bit := 6;
   // "3Fok_2".ADDR_Bit := 7;
   // "3Fok_sh".ADDR_Byte := 1;
   // "3Fok_sh".ADDR_Bit := 0;
   // SHUSKV_Ok.ADDR_Byte := 1;
   // SHUSKV_Ok.ADDR_Bit := 1;
   // Leak_KP_res.ADDR_Byte := 1;
   // Leak_KP_res.ADDR_Bit := 2;
   // Leak_KP_res_1.ADDR_Byte := 1;
   // Leak_KP_res_1.ADDR_Bit := 3;
   VAR_TEMP   // added for the SCL form of the ladder/FBD networks
      _w1 : Bool;
   END_VAR
BEGIN

REGION Network 1: AllBlock
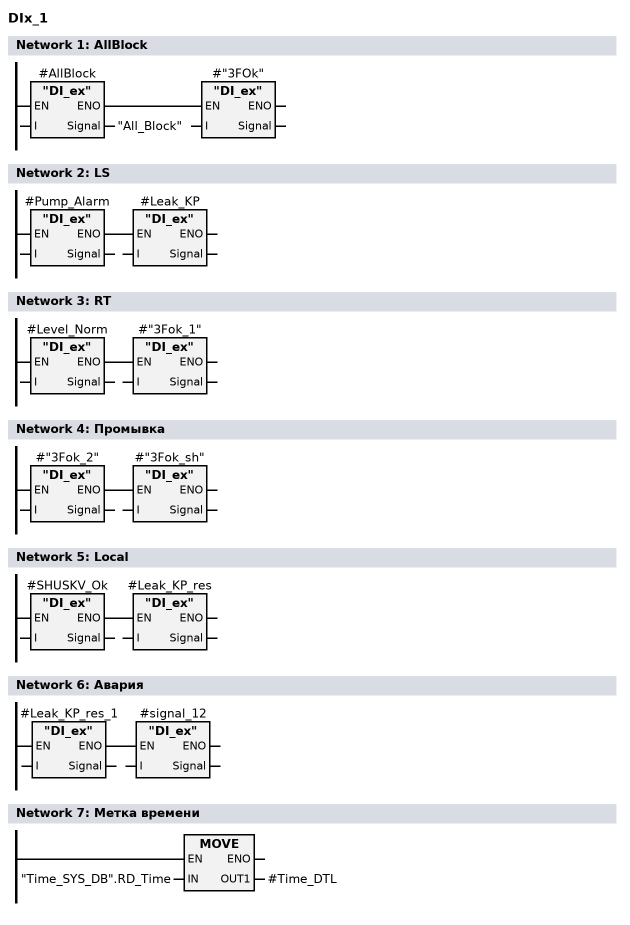
   RUNG wire#powerrail
      #AllBlock(I :=, Signal => "All_Block")
      #"3FOk"(I :=, Signal =>)
   END_RUNG
   // the same network as SCL:
   #AllBlock(Signal => "All_Block", ENO => #_w1);   // "DI_ex"
   IF #_w1 THEN
       #"3FOk"();   // "DI_ex"
   END_IF;
END_REGION

REGION Network 2: LS
   RUNG wire#powerrail
      #Pump_Alarm(I :=, Signal =>)
      #Leak_KP(I :=, Signal =>)
   END_RUNG
   // the same network as SCL:
   #Pump_Alarm(ENO => #_w1);   // "DI_ex"
   IF #_w1 THEN
       #Leak_KP();   // "DI_ex"
   END_IF;
END_REGION

REGION Network 3: RT
   RUNG wire#powerrail
      #Level_Norm(I :=, Signal =>)
      #"3Fok_1"(I :=, Signal =>)
   END_RUNG
   // the same network as SCL:
   #Level_Norm(ENO => #_w1);   // "DI_ex"
   IF #_w1 THEN
       #"3Fok_1"();   // "DI_ex"
   END_IF;
END_REGION

REGION Network 4: Промывка
   RUNG wire#powerrail
      #"3Fok_2"(I :=, Signal =>)
      #"3Fok_sh"(I :=, Signal =>)
   END_RUNG
   // the same network as SCL:
   #"3Fok_2"(ENO => #_w1);   // "DI_ex"
   IF #_w1 THEN
       #"3Fok_sh"();   // "DI_ex"
   END_IF;
END_REGION

REGION Network 5: Local
   RUNG wire#powerrail
      #SHUSKV_Ok(I :=, Signal =>)
      #Leak_KP_res(I :=, Signal =>)
   END_RUNG
   // the same network as SCL:
   #SHUSKV_Ok(ENO => #_w1);   // "DI_ex"
   IF #_w1 THEN
       #Leak_KP_res();   // "DI_ex"
   END_IF;
END_REGION

REGION Network 6: Авария
   RUNG wire#powerrail
      #Leak_KP_res_1(I :=, Signal =>)
      #signal_12(I :=, Signal =>)
   END_RUNG
   // the same network as SCL:
   #Leak_KP_res_1(ENO => #_w1);   // "DI_ex"
   IF #_w1 THEN
       #signal_12();   // "DI_ex"
   END_IF;
END_REGION

REGION Network 7: Метка времени
   RUNG wire#powerrail
      Move(in := "Time_SYS_DB".RD_Time, out1 => #Time_DTL)
   END_RUNG
   // the same network as SCL:
   #Time_DTL := "Time_SYS_DB".RD_Time;
END_REGION
END_FUNCTION_BLOCK

FUNCTION_BLOCK "DI_ex"   // FB101, LAD
{ S7_Optimized_Access := 'FALSE' }
VERSION : 0.1
// stored: AutoNumber false, IsIECCheckEnabled false, SetENOAutomatically false, UDAEnableTagReadback false
   VAR_INPUT
      I : Bool;   // Входной сигнал ПЛК
   END_VAR
   VAR_OUTPUT
      Signal : Bool;   // Результат обработки
   END_VAR
   VAR DB_SPECIFIC
      CMD : "CMD";   // Основные команды / Блок команд
      Use : Struct
         Inverse { S7_SetPoint := 'True'} : Bool;   // Инверсия входного сигнала
         Indirect { S7_SetPoint := 'True'} : Bool := true;   // Использование косвенной адресации
      END_STRUCT;
      ADDR_Byte { S7_SetPoint := 'True'} : Int;   // Адрес входа на контроллере (Байт)
      ADDR_Bit { S7_SetPoint := 'True'} : Int := 9;   // Адрес входа на контроллере (Бит)
   END_VAR
   VAR
      Filter_On { S7_SetPoint := 'True'} : "Time_S_b";   // Фильтр наличия сигнала
      Filter_Off { S7_SetPoint := 'True'} : "Time_S_b";   // Фильтр отсутствия сигнала
   END_VAR
   VAR_TEMP
      Data : Bool;
   END_VAR
   VAR_TEMP   // added for the SCL form of the ladder/FBD networks
      _w1 : Bool;
      _w2 : Bool;
   END_VAR
BEGIN

REGION Network 1: Устройство в ручном режиме
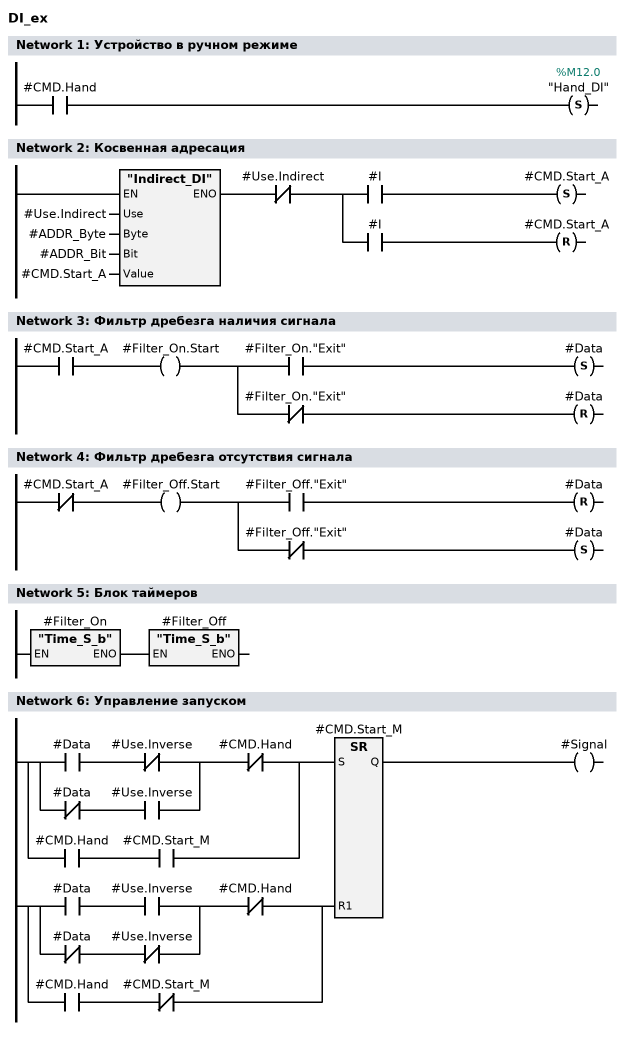
   RUNG wire#powerrail
      Contact( #CMD.Hand )
      S_Coil( "Hand_DI" )
   END_RUNG
   // the same network as SCL:
   IF #CMD.Hand THEN "Hand_DI" := TRUE; END_IF;
END_REGION

REGION Network 2: Косвенная адресация
   RUNG wire#powerrail
      "Indirect_DI"(Use := #Use.Indirect, "Byte" := #ADDR_Byte, Bit := #ADDR_Bit, Value := #CMD.Start_A)
      I_Contact( #Use.Indirect )
      wire#w1
      Contact( #I )
      S_Coil( #CMD.Start_A )
   END_RUNG
   RUNG wire#w1
      Contact( #I )
      R_Coil( #CMD.Start_A )
   END_RUNG
   // the same network as SCL:
   "Indirect_DI"(Use := #Use.Indirect,
                 "Byte" := #ADDR_Byte,
                 Bit := #ADDR_Bit,
                 Value := #CMD.Start_A,
                 ENO => #_w1);
   #_w2 := #_w1 AND NOT #Use.Indirect;
   IF #_w2 AND #I THEN
       #CMD.Start_A := TRUE;
       #CMD.Start_A := FALSE;
   END_IF;
END_REGION

REGION Network 3: Фильтр дребезга наличия сигнала
   RUNG wire#powerrail
      Contact( #CMD.Start_A )
      Coil( #Filter_On.Start )
      wire#w1
      Contact( #Filter_On."Exit" )
      S_Coil( #Data )
   END_RUNG
   RUNG wire#w1
      I_Contact( #Filter_On."Exit" )
      R_Coil( #Data )
   END_RUNG
   // the same network as SCL:
   #Filter_On.Start := #CMD.Start_A;
   IF #CMD.Start_A AND #Filter_On."Exit" THEN #Data := TRUE; END_IF;
   IF #CMD.Start_A AND NOT #Filter_On."Exit" THEN #Data := FALSE; END_IF;
END_REGION

REGION Network 4: Фильтр дребезга отсутствия сигнала
   RUNG wire#powerrail
      I_Contact( #CMD.Start_A )
      Coil( #Filter_Off.Start )
      wire#w1
      Contact( #Filter_Off."Exit" )
      R_Coil( #Data )
   END_RUNG
   RUNG wire#w1
      I_Contact( #Filter_Off."Exit" )
      S_Coil( #Data )
   END_RUNG
   // the same network as SCL:
   #Filter_Off.Start := NOT #CMD.Start_A;
   IF NOT #CMD.Start_A AND #Filter_Off."Exit" THEN #Data := FALSE; END_IF;
   IF NOT #CMD.Start_A AND NOT #Filter_Off."Exit" THEN #Data := TRUE; END_IF;
END_REGION

REGION Network 5: Блок таймеров
   RUNG wire#powerrail
      #Filter_On()
      #Filter_Off()
   END_RUNG
   // the same network as SCL:
   #Filter_On(ENO => #_w1);   // "Time_S_b"
   IF #_w1 THEN
       #Filter_Off();   // "Time_S_b"
   END_IF;
END_REGION

REGION Network 6: Управление запуском
   RUNG wire#powerrail
      Contact( #Data )
      I_Contact( #Use.Inverse )
      wire#w1
      I_Contact( #CMD.Hand )
      wire#w2
      S_SR(operand := #CMD.Start_M, r1 := wire#w4)
      Coil( #Signal )
   END_RUNG
   RUNG wire#powerrail
      I_Contact( #Data )
      Contact( #Use.Inverse )
   END_RUNG wire#w1
   RUNG wire#powerrail
      Contact( #CMD.Hand )
      Contact( #CMD.Start_M )
   END_RUNG wire#w2
   RUNG wire#powerrail
      Contact( #Data )
      Contact( #Use.Inverse )
      wire#w3
      I_Contact( #CMD.Hand )
   END_RUNG wire#w4
   RUNG wire#powerrail
      I_Contact( #Data )
      I_Contact( #Use.Inverse )
   END_RUNG wire#w3
   RUNG wire#powerrail
      Contact( #CMD.Hand )
      I_Contact( #CMD.Start_M )
   END_RUNG wire#w4
   // the same network as SCL:
   #_w1 := (((#Data AND #Use.Inverse) OR (NOT #Data AND NOT #Use.Inverse)) AND NOT #CMD.Hand) OR (#CMD.Hand AND NOT #CMD.Start_M);
   IF (((#Data AND NOT #Use.Inverse) OR (NOT #Data AND #Use.Inverse)) AND NOT #CMD.Hand) OR (#CMD.Hand AND #CMD.Start_M) THEN
       #CMD.Start_M := TRUE;   // SR flip-flop
   END_IF;
   IF #_w1 THEN #CMD.Start_M := FALSE; END_IF;
   #Signal := #CMD.Start_M;
END_REGION
END_FUNCTION_BLOCK

FUNCTION_BLOCK "Time_S_b"   // FB89, LAD
{ S7_Optimized_Access := 'FALSE' }
VERSION : 0.1
// stored: AutoNumber false, IsIECCheckEnabled false, SetENOAutomatically false, UDAEnableTagReadback false
   VAR DB_SPECIFIC
      SP { S7_SetPoint := 'True'} : Byte := 2;   // Уставка
      Now : Byte;   // Текущий счёт
      Start : Bool;   // Запуск
      "Exit" : Bool;   // Счёт завершён
      Pause : Bool;   // Пауза
      Reset : Bool;   // Сброс таймера
   END_VAR
   VAR_TEMP   // added for the SCL form of the ladder/FBD networks
      _w1 : Bool;
   END_VAR
BEGIN

REGION Network 1: Подсчёт времени
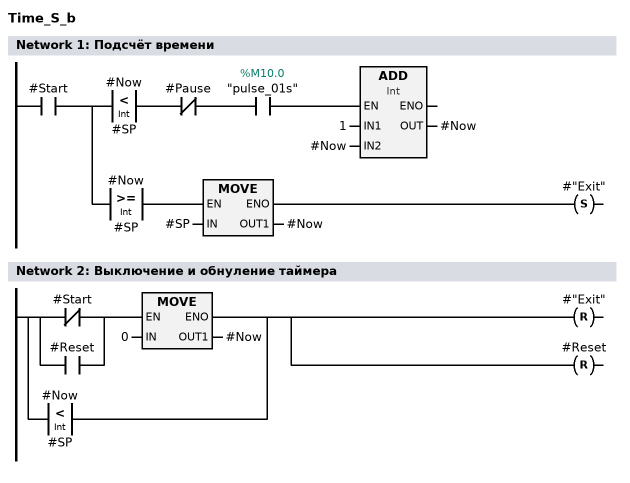
   RUNG wire#powerrail
      Contact( #Start )
      wire#w1
      { S7_Templates := "SrcType := Int" } LT_Contact(in1 := #Now, in2 := #SP)
      I_Contact( #Pause )
      Contact( "pulse_01s" )
      { S7_Templates := "SrcType := Int"; S7_GenerateENO := "TRUE" } Add(in1 := 1, in2 := #Now, out => #Now)
   END_RUNG
   RUNG wire#w1
      { S7_Templates := "SrcType := Int" } GE_Contact(in1 := #Now, in2 := #SP)
      { S7_GenerateENO := "TRUE" } Move(in := #SP, out1 => #Now)
      S_Coil( #"Exit" )
   END_RUNG
   // the same network as SCL:
   // ENO of a box is taken as its EN; it also drops when the box reports an error
   IF #Start AND (#Now < #SP) AND NOT #Pause AND "pulse_01s" THEN #Now := 1 + #Now; END_IF;
   #_w1 := #Start AND (#Now >= #SP);
   IF #_w1 THEN
       #Now := #SP;
       #"Exit" := TRUE;
   END_IF;
END_REGION

REGION Network 2: Выключение и обнуление таймера
   RUNG wire#powerrail
      I_Contact( #Start )
      wire#w1
      { S7_GenerateENO := "TRUE" } Move(in := 0, out1 => #Now)
      wire#w2
      R_Coil( #"Exit" )
   END_RUNG
   RUNG wire#powerrail
      Contact( #Reset )
   END_RUNG wire#w1
   RUNG wire#powerrail
      { S7_Templates := "SrcType := Int" } LT_Contact(in1 := #Now, in2 := #SP)
   END_RUNG wire#w2
   RUNG wire#w2
      R_Coil( #Reset )
   END_RUNG
   // the same network as SCL:
   // ENO of a box is taken as its EN; it also drops when the box reports an error
   #_w1 := NOT #Start OR #Reset;
   IF #_w1 THEN #Now := 0; END_IF;
   IF #_w1 OR (#Now < #SP) THEN
       #"Exit" := FALSE;
       #Reset := FALSE;
   END_IF;
END_REGION
END_FUNCTION_BLOCK

FUNCTION_BLOCK "AIx"   // FB220, LAD
{ S7_Optimized_Access := 'FALSE' }
VERSION : 0.1
// Signal - PIW код сигнала от датчика
// pulse - частота алгоритма фильтрации
// Result - результат обработки сигнала, формат Real
// stored: AutoNumber false, IsIECCheckEnabled false, SetENOAutomatically false, UDAEnableTagReadback false
   VAR DB_SPECIFIC
      Time_DTL { S7_SetPoint := 'True'} : DTL;
   END_VAR
   VAR_TEMP   // added for the SCL form of the ladder/FBD networks
      _w1 : Bool;
      _w2 : Bool;
   END_VAR
BEGIN

REGION Network 1: Датчик уровня
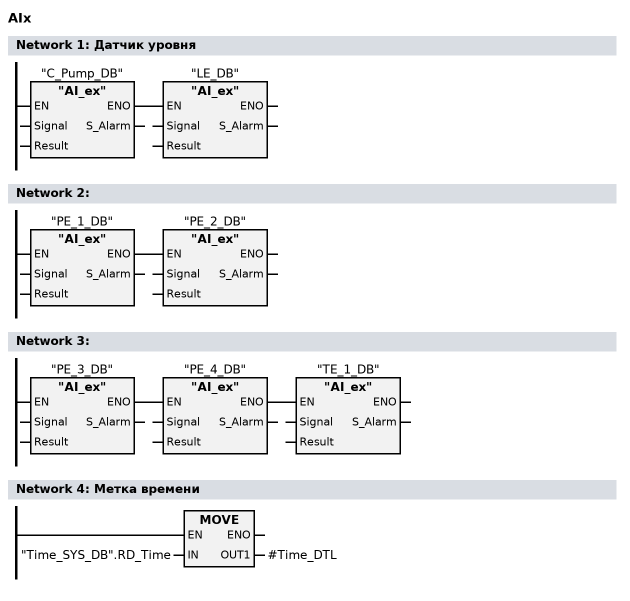
   RUNG wire#powerrail
      "C_Pump_DB"(Signal :=, Result :=, S_Alarm =>)
      "LE_DB"(Signal :=, Result :=, S_Alarm =>)
   END_RUNG
   // the same network as SCL:
   "C_Pump_DB"(ENO => #_w1);   // "AI_ex"
   IF #_w1 THEN
       "LE_DB"();   // "AI_ex"
   END_IF;
END_REGION

REGION Network 2
   RUNG wire#powerrail
      "PE_1_DB"(Signal :=, Result :=, S_Alarm =>)
      "PE_2_DB"(Signal :=, Result :=, S_Alarm =>)
   END_RUNG
   // the same network as SCL:
   "PE_1_DB"(ENO => #_w1);   // "AI_ex"
   IF #_w1 THEN
       "PE_2_DB"();   // "AI_ex"
   END_IF;
END_REGION

REGION Network 3
   RUNG wire#powerrail
      "PE_3_DB"(Signal :=, Result :=, S_Alarm =>)
      "PE_4_DB"(Signal :=, Result :=, S_Alarm =>)
      "TE_1_DB"(Signal :=, Result :=, S_Alarm =>)
   END_RUNG
   // the same network as SCL:
   "PE_3_DB"(ENO => #_w1);   // "AI_ex"
   "PE_4_DB"(EN := #_w1, ENO => #_w2);   // "AI_ex"
   IF #_w2 THEN
       "TE_1_DB"();   // "AI_ex"
   END_IF;
END_REGION

REGION Network 4: Метка времени
   RUNG wire#powerrail
      Move(in := "Time_SYS_DB".RD_Time, out1 => #Time_DTL)
   END_RUNG
   // the same network as SCL:
   #Time_DTL := "Time_SYS_DB".RD_Time;
END_REGION
END_FUNCTION_BLOCK

FUNCTION_BLOCK "AI_ex"   // FB103, LAD
{ S7_Optimized_Access := 'FALSE' }
VERSION : 0.1
// stored: AutoNumber false, IsIECCheckEnabled false, SetENOAutomatically false, UDAEnableTagReadback false
   VAR_OUTPUT
      S_Alarm : Bool;   // Внешний индикатор наличия аварии
   END_VAR
   VAR_IN_OUT
      Signal : Int;   // Входной сигнал контроллера
      Result : Real;   // Результат измерений
   END_VAR
   VAR DB_SPECIFIC
      CMD : "CMD";   // Основные команды / Блок команд
      Mode : Int;   // Режим работы
      Status : Int;   // Статус устройства
      Use : Struct   // Функционал
         RTD { S7_SetPoint := 'True'} : Bool;   // Режим RTD
         Filter { S7_SetPoint := 'True'} : Bool;   // Филтрация сигнала
         Inverse { S7_SetPoint := 'True'} : Bool;   // Инверсия сигнала
         Indirect { S7_SetPoint := 'True'} : Bool := true;   // Косвенная адресация
         Status { S7_SetPoint := 'True'} : Bool;   // Использовать подсветку
         Light { S7_SetPoint := 'True'} : Bool;   // Динамическая подсветка
         Lim_Low { S7_SetPoint := 'True'} : Bool;   // Отсечь низкие аварии
         Lim_High { S7_SetPoint := 'True'} : Bool;   // Отсечь высокие аварии
         Communication { S7_SetPoint := 'True'} : Bool;   // Передача в Value по сети
      END_STRUCT;
      VmA : Real;   // Реальный сигнал на входе ПЛК
      RTD_c { S7_SetPoint := 'True'} : Real := 10.0;   // Коэффициент RTD
      Calibration { S7_SetPoint := 'True'} : Real;   // Поправка
   END_VAR
   VAR
      Converter { S7_SetPoint := 'True'} : "Converter_LAD";   // Масштабирование сигнала
   END_VAR
   VAR DB_SPECIFIC
      SP : Struct   // Уставки аварий
         NC { S7_SetPoint := 'True'} : Real := -500.0;   // Сигнал при обрыве линии
         SC { S7_SetPoint := 'True'} : Real := 32000.0;   // Сигнал при КЗ/перегрузке
         HH { S7_SetPoint := 'True'} : Real := 90.0;   // Аварийно высокий сигнал
         H { S7_SetPoint := 'True'} : Real := 85.0;   // Высокий сигнал
         L { S7_SetPoint := 'True'} : Real := 15.0;   // Низкий сигнал
         LL { S7_SetPoint := 'True'} : Real := 10.0;   // Аварийно низкий сигнал
      END_STRUCT;
   END_VAR
   VAR
      Tx { S7_SetPoint := 'True'} : Array[0..5] of "Time_R";   // Блок таймеров
   END_VAR
   VAR DB_SPECIFIC
      Alarm : Struct   // Список аварий
         ST : Bool;   // Общая неисправность
         HH : Bool;   // сработала авария по аварийно высокму уровню
         H : Bool;   // сработало предупреждение по высокому уровню
         L : Bool;   // сработало предупреждение по низкому уровню
         LL : Bool;   // сработало предупрждение по аварийно низкому уровню
         NC : Bool;   // обрыв линии
         SC : Bool;   // короткое замыкание
      END_STRUCT;
      Alarms : Word;   // Слово аварий
      Events : Word;   // События датчика
      pos : Array[0..15] of Bool;   // Контроль фронтов событий
      Input_Type { S7_SetPoint := 'True'} : Int;   // Тип датчика, 0 - 4..20, 1 - 0..20, 2 - 0..10, 3 - 0..5, 4 - RTD
      CodeID { S7_SetPoint := 'True'} : Int;   // Код датчика для привязки в скаде
      "Type" { S7_SetPoint := 'True'} : Int;   // Тип датчика (единицы измерения)
      ADDR { S7_SetPoint := 'True'} : Int;   // Адрес входа на контроллере
      Filter_SP { S7_SetPoint := 'True'} : Int := 100;   // Ёмкость фильтра
      "Name" { S7_SetPoint := 'True'} : String[5];
   END_VAR
   VAR
      Filter_DB : "Filter";   // Фильтрация скачков сигнала
   END_VAR
   VAR DB_SPECIFIC
      Time_DTL { S7_SetPoint := 'True'} : DTL;
   END_VAR
   VAR_TEMP
      ev : Bool;   // Флаг событий
      Value : Real;   // Итоговый сигнал
      Signal_DI : DInt;   // Конвертация сигнала
      Signal_R : Real;   // Конвертация сигнала
      Type_Min : Real;
      Type_Max : Real;
   END_VAR
   VAR CONSTANT
      FALSE : Bool;
      TRUE : Bool := true;
   END_VAR
   // CMD.Start_A := true;
   // Converter.Max_In := 27648.0;
   // Converter.Max_Out := 100.0;
   VAR_TEMP   // added for the SCL form of the ladder/FBD networks
      _w1 : Bool;
      _w2 : Bool;
      _w3 : Bool;
      _w4 : Bool;
      _w5 : Bool;
      _w6 : Bool;
      _w7 : Bool;
      _w8 : Bool;
      _w9 : Bool;
      _w10 : Bool;
      _w11 : Bool;
      _w12 : Bool;
      _w13 : Bool;
      _w14 : Bool;
      _w15 : Bool;
      _w16 : Bool;
   END_VAR
BEGIN

REGION Network 1: Общий сброс
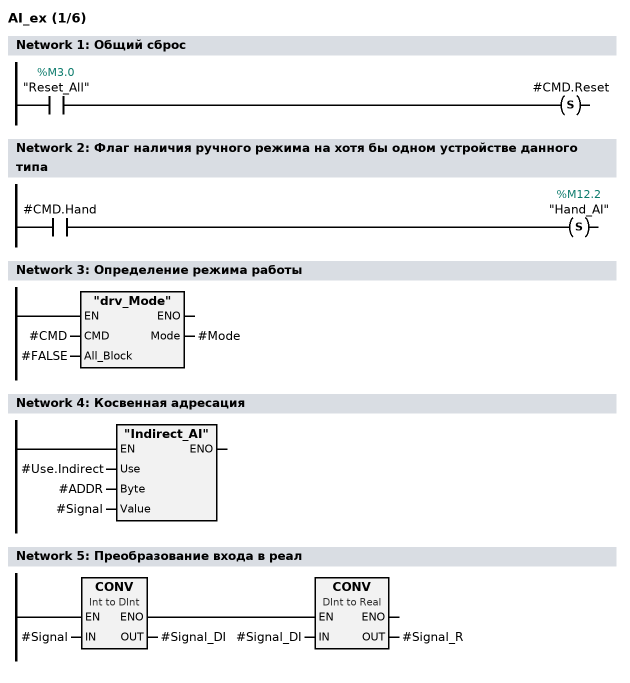
   RUNG wire#powerrail
      Contact( "Reset_All" )
      S_Coil( #CMD.Reset )
   END_RUNG
   // the same network as SCL:
   IF "Reset_All" THEN #CMD.Reset := TRUE; END_IF;
END_REGION

REGION Network 2: Флаг наличия ручного режима на хотя бы одном устройстве данного типа
   RUNG wire#powerrail
      Contact( #CMD.Hand )
      S_Coil( "Hand_AI" )
   END_RUNG
   // the same network as SCL:
   IF #CMD.Hand THEN "Hand_AI" := TRUE; END_IF;
END_REGION

REGION Network 3: Определение режима работы
   RUNG wire#powerrail
      "drv_Mode"(CMD := #CMD, All_Block := #FALSE, Mode => #Mode)
   END_RUNG
   // the same network as SCL:
   "drv_Mode"(CMD := #CMD, All_Block := #FALSE, Mode => #Mode);
END_REGION

REGION Network 4: Косвенная адресация
   RUNG wire#powerrail
      "Indirect_AI"(Use := #Use.Indirect, "Byte" := #ADDR, Value := #Signal)
   END_RUNG
   // the same network as SCL:
   "Indirect_AI"(Use := #Use.Indirect, "Byte" := #ADDR, Value := #Signal);
END_REGION

REGION Network 5: Преобразование входа в реал
   RUNG wire#powerrail
      { S7_Templates := "[SrcType := Int, DestType := DInt]"; S7_GenerateENO := "TRUE" } Convert(in := #Signal, out => #Signal_DI)
      { S7_Templates := "[SrcType := DInt, DestType := Real]"; S7_GenerateENO := "TRUE" } Convert(in := #Signal_DI, out => #Signal_R)
   END_RUNG
   // the same network as SCL:
   // ENO of a box is taken as its EN; it also drops when the box reports an error
   #Signal_DI := INT_TO_DINT(#Signal);
   #Signal_R := DINT_TO_REAL(#Signal_DI);
END_REGION

REGION Network 6: Преобразование кода в реальное значение входа
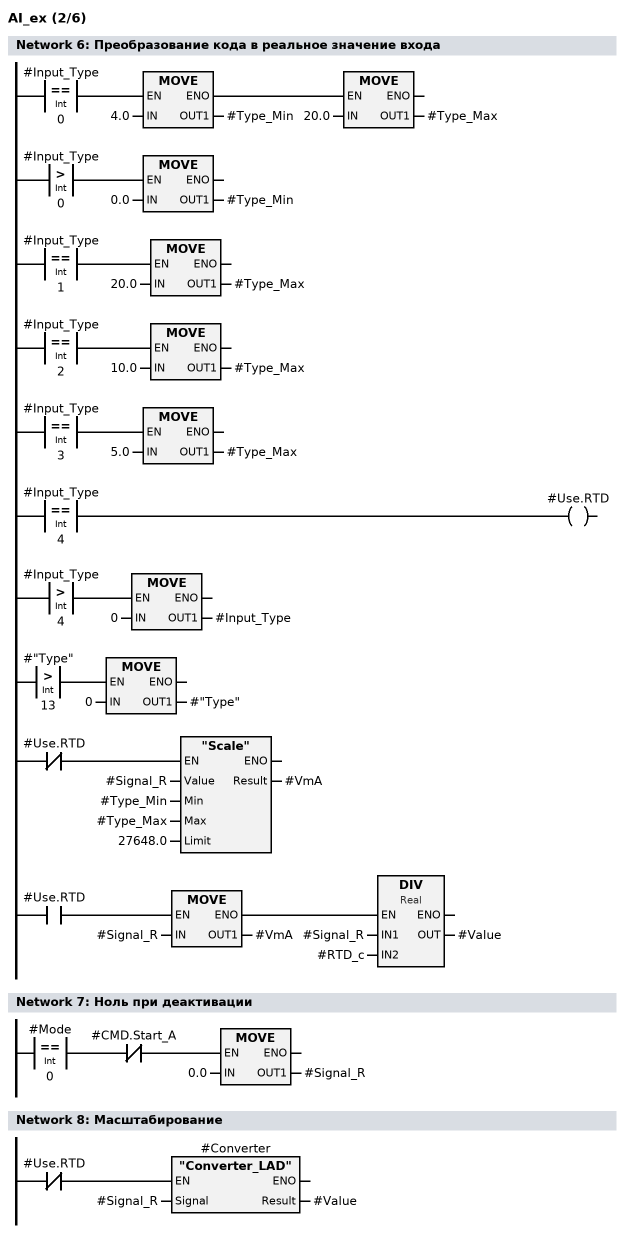
   RUNG wire#powerrail
      { S7_Templates := "SrcType := Int" } EQ_Contact(in1 := #Input_Type, in2 := 0)
      Move(in := 4.0, out1 => #Type_Min)
      Move(in := 20.0, out1 => #Type_Max)
   END_RUNG
   RUNG wire#powerrail
      { S7_Templates := "SrcType := Int" } GT_Contact(in1 := #Input_Type, in2 := 0)
      Move(in := 0.0, out1 => #Type_Min)
   END_RUNG
   RUNG wire#powerrail
      { S7_Templates := "SrcType := Int" } EQ_Contact(in1 := #Input_Type, in2 := 1)
      Move(in := 20.0, out1 => #Type_Max)
   END_RUNG
   RUNG wire#powerrail
      { S7_Templates := "SrcType := Int" } EQ_Contact(in1 := #Input_Type, in2 := 2)
      Move(in := 10.0, out1 => #Type_Max)
   END_RUNG
   RUNG wire#powerrail
      { S7_Templates := "SrcType := Int" } EQ_Contact(in1 := #Input_Type, in2 := 3)
      Move(in := 5.0, out1 => #Type_Max)
   END_RUNG
   RUNG wire#powerrail
      { S7_Templates := "SrcType := Int" } EQ_Contact(in1 := #Input_Type, in2 := 4)
      Coil( #Use.RTD )
   END_RUNG
   RUNG wire#powerrail
      { S7_Templates := "SrcType := Int" } GT_Contact(in1 := #Input_Type, in2 := 4)
      Move(in := 0, out1 => #Input_Type)
   END_RUNG
   RUNG wire#powerrail
      { S7_Templates := "SrcType := Int" } GT_Contact(in1 := #"Type", in2 := 13)
      Move(in := 0, out1 => #"Type")
   END_RUNG
   RUNG wire#powerrail
      I_Contact( #Use.RTD )
      "Scale"(Value := #Signal_R, Min := #Type_Min, Max := #Type_Max, Limit := 27648.0, Result => #VmA)
   END_RUNG
   RUNG wire#powerrail
      Contact( #Use.RTD )
      Move(in := #Signal_R, out1 => #VmA)
      { S7_Templates := "SrcType := Real"; S7_GenerateENO := "TRUE" } Div(in1 := #Signal_R, in2 := #RTD_c, out => #Value)
   END_RUNG
   // the same network as SCL:
   IF #Input_Type = 0 THEN
       #Type_Min := 4.0;
       #Type_Max := 20.0;
   END_IF;
   IF #Input_Type > 0 THEN #Type_Min := 0.0; END_IF;
   IF #Input_Type = 1 THEN #Type_Max := 20.0; END_IF;
   IF #Input_Type = 2 THEN #Type_Max := 10.0; END_IF;
   IF #Input_Type = 3 THEN #Type_Max := 5.0; END_IF;
   #Use.RTD := #Input_Type = 4;
   IF #Input_Type > 4 THEN #Input_Type := 0; END_IF;
   IF #"Type" > 13 THEN #"Type" := 0; END_IF;
   IF NOT #Use.RTD THEN
       "Scale"(Value := #Signal_R, Min := #Type_Min, Max := #Type_Max, Limit := 27648.0, Result => #VmA);
   END_IF;
   IF #Use.RTD THEN
       #VmA := #Signal_R;
       #Value := #Signal_R / #RTD_c;
   END_IF;
END_REGION

REGION Network 7: Ноль при деактивации
   RUNG wire#powerrail
      { S7_Templates := "SrcType := Int" } EQ_Contact(in1 := #Mode, in2 := 0)
      I_Contact( #CMD.Start_A )
      Move(in := 0.0, out1 => #Signal_R)
   END_RUNG
   // the same network as SCL:
   IF (#Mode = 0) AND NOT #CMD.Start_A THEN #Signal_R := 0.0; END_IF;
END_REGION

REGION Network 8: Масштабирование
   RUNG wire#powerrail
      I_Contact( #Use.RTD )
      #Converter(Signal := #Signal_R, Result => #Value)
   END_RUNG
   // the same network as SCL:
   IF NOT #Use.RTD THEN
       #Converter(Signal := #Signal_R, Result => #Value);   // "Converter_LAD"
   END_IF;
END_REGION

REGION Network 9: Вызов блока фильтрации
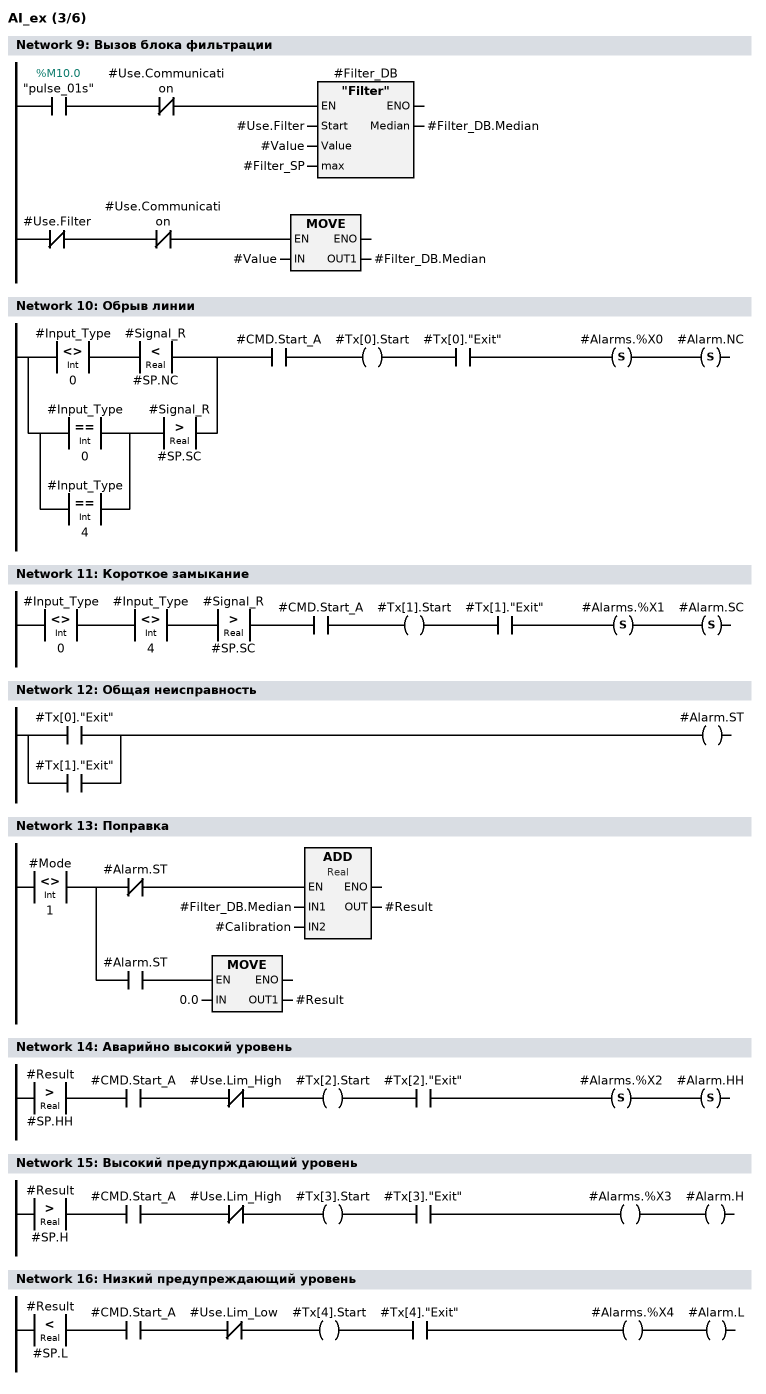
   RUNG wire#powerrail
      Contact( "pulse_01s" )
      I_Contact( #Use.Communication )
      #Filter_DB(Start := #Use.Filter, Value := #Value, max := #Filter_SP, Median => #Filter_DB.Median)
   END_RUNG
   RUNG wire#powerrail
      I_Contact( #Use.Filter )
      I_Contact( #Use.Communication )
      { S7_GenerateENO := "TRUE" } Move(in := #Value, out1 => #Filter_DB.Median)
   END_RUNG
   // the same network as SCL:
   IF "pulse_01s" AND NOT #Use.Communication THEN
       #Filter_DB(Start := #Use.Filter, Value := #Value, max := #Filter_SP, Median => #Filter_DB.Median);   // "Filter"
   END_IF;
   IF NOT #Use.Filter AND NOT #Use.Communication THEN #Filter_DB.Median := #Value; END_IF;
END_REGION

REGION Network 10: Обрыв линии
   RUNG wire#powerrail
      { S7_Templates := "SrcType := Int" } NE_Contact(in1 := #Input_Type, in2 := 0)
      { S7_Templates := "SrcType := Real" } LT_Contact(in1 := #Signal_R, in2 := #SP.NC)
      wire#w1
      Contact( #CMD.Start_A )
      Coil( #Tx[0].Start )
      Contact( #Tx[0]."Exit" )
      S_Coil( #Alarms.%X0 )
      S_Coil( #Alarm.NC )
   END_RUNG
   RUNG wire#powerrail
      { S7_Templates := "SrcType := Int" } EQ_Contact(in1 := #Input_Type, in2 := 0)
      wire#w2
      { S7_Templates := "SrcType := Real" } GT_Contact(in1 := #Signal_R, in2 := #SP.SC)
   END_RUNG wire#w1
   RUNG wire#powerrail
      { S7_Templates := "SrcType := Int" } EQ_Contact(in1 := #Input_Type, in2 := 4)
   END_RUNG wire#w2
   // the same network as SCL:
   #Tx[0].Start := (((#Input_Type <> 0) AND (#Signal_R < #SP.NC)) OR (((#Input_Type = 0) OR (#Input_Type = 4)) AND (#Signal_R > #SP.SC))) AND #CMD.Start_A;
   IF (((#Input_Type <> 0) AND (#Signal_R < #SP.NC)) OR (((#Input_Type = 0) OR (#Input_Type = 4)) AND (#Signal_R > #SP.SC))) AND #CMD.Start_A AND #Tx[0]."Exit" THEN
       #Alarms.%X0 := TRUE;
       #Alarm.NC := TRUE;
   END_IF;
END_REGION

REGION Network 11: Короткое замыкание
   RUNG wire#powerrail
      { S7_Templates := "SrcType := Int" } NE_Contact(in1 := #Input_Type, in2 := 0)
      { S7_Templates := "SrcType := Int" } NE_Contact(in1 := #Input_Type, in2 := 4)
      { S7_Templates := "SrcType := Real" } GT_Contact(in1 := #Signal_R, in2 := #SP.SC)
      Contact( #CMD.Start_A )
      Coil( #Tx[1].Start )
      Contact( #Tx[1]."Exit" )
      S_Coil( #Alarms.%X1 )
      S_Coil( #Alarm.SC )
   END_RUNG
   // the same network as SCL:
   #Tx[1].Start := (#Input_Type <> 0) AND (#Input_Type <> 4) AND (#Signal_R > #SP.SC) AND #CMD.Start_A;
   IF (#Input_Type <> 0) AND (#Input_Type <> 4) AND (#Signal_R > #SP.SC) AND #CMD.Start_A AND #Tx[1]."Exit" THEN
       #Alarms.%X1 := TRUE;
       #Alarm.SC := TRUE;
   END_IF;
END_REGION

REGION Network 12: Общая неисправность
   RUNG wire#powerrail
      Contact( #Tx[0]."Exit" )
      wire#w1
      Coil( #Alarm.ST )
   END_RUNG
   RUNG wire#powerrail
      Contact( #Tx[1]."Exit" )
   END_RUNG wire#w1
   // the same network as SCL:
   #Alarm.ST := #Tx[0]."Exit" OR #Tx[1]."Exit";
END_REGION

REGION Network 13: Поправка
   RUNG wire#powerrail
      { S7_Templates := "SrcType := Int" } NE_Contact(in1 := #Mode, in2 := 1)
      wire#w1
      I_Contact( #Alarm.ST )
      { S7_Templates := "SrcType := Real"; S7_GenerateENO := "TRUE" } Add(in1 := #Filter_DB.Median, in2 := #Calibration, out => #Result)
   END_RUNG
   RUNG wire#w1
      Contact( #Alarm.ST )
      Move(in := 0.0, out1 => #Result)
   END_RUNG
   // the same network as SCL:
   #_w1 := #Mode <> 1;
   IF #_w1 AND NOT #Alarm.ST THEN #Result := #Filter_DB.Median + #Calibration; END_IF;
   IF #_w1 AND #Alarm.ST THEN #Result := 0.0; END_IF;
END_REGION

REGION Network 14: Аварийно высокий уровень
   RUNG wire#powerrail
      { S7_Templates := "SrcType := Real" } GT_Contact(in1 := #Result, in2 := #SP.HH)
      Contact( #CMD.Start_A )
      I_Contact( #Use.Lim_High )
      Coil( #Tx[2].Start )
      Contact( #Tx[2]."Exit" )
      S_Coil( #Alarms.%X2 )
      S_Coil( #Alarm.HH )
   END_RUNG
   // the same network as SCL:
   #Tx[2].Start := (#Result > #SP.HH) AND #CMD.Start_A AND NOT #Use.Lim_High;
   IF (#Result > #SP.HH) AND #CMD.Start_A AND NOT #Use.Lim_High AND #Tx[2]."Exit" THEN
       #Alarms.%X2 := TRUE;
       #Alarm.HH := TRUE;
   END_IF;
END_REGION

REGION Network 15: Высокий предупрждающий уровень
   RUNG wire#powerrail
      { S7_Templates := "SrcType := Real" } GT_Contact(in1 := #Result, in2 := #SP.H)
      Contact( #CMD.Start_A )
      I_Contact( #Use.Lim_High )
      Coil( #Tx[3].Start )
      Contact( #Tx[3]."Exit" )
      Coil( #Alarms.%X3 )
      Coil( #Alarm.H )
   END_RUNG
   // the same network as SCL:
   #Tx[3].Start := (#Result > #SP.H) AND #CMD.Start_A AND NOT #Use.Lim_High;
   #Alarms.%X3 := (#Result > #SP.H) AND #CMD.Start_A AND NOT #Use.Lim_High AND #Tx[3]."Exit";
   #Alarm.H := #Alarms.%X3;
END_REGION

REGION Network 16: Низкий предупреждающий уровень
   RUNG wire#powerrail
      { S7_Templates := "SrcType := Real" } LT_Contact(in1 := #Result, in2 := #SP.L)
      Contact( #CMD.Start_A )
      I_Contact( #Use.Lim_Low )
      Coil( #Tx[4].Start )
      Contact( #Tx[4]."Exit" )
      Coil( #Alarms.%X4 )
      Coil( #Alarm.L )
   END_RUNG
   // the same network as SCL:
   #Tx[4].Start := (#Result < #SP.L) AND #CMD.Start_A AND NOT #Use.Lim_Low;
   #Alarms.%X4 := (#Result < #SP.L) AND #CMD.Start_A AND NOT #Use.Lim_Low AND #Tx[4]."Exit";
   #Alarm.L := #Alarms.%X4;
END_REGION

REGION Network 17: Аварийно высокий уровень
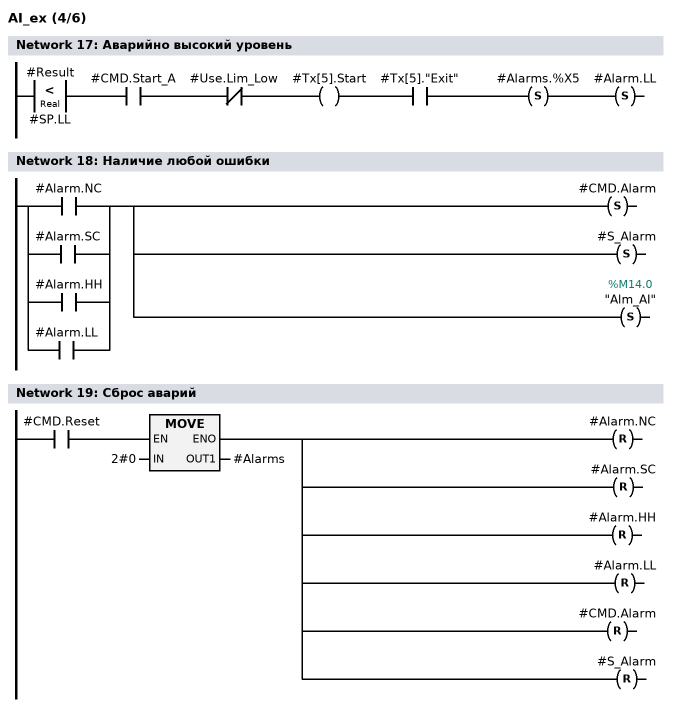
   RUNG wire#powerrail
      { S7_Templates := "SrcType := Real" } LT_Contact(in1 := #Result, in2 := #SP.LL)
      Contact( #CMD.Start_A )
      I_Contact( #Use.Lim_Low )
      Coil( #Tx[5].Start )
      Contact( #Tx[5]."Exit" )
      S_Coil( #Alarms.%X5 )
      S_Coil( #Alarm.LL )
   END_RUNG
   // the same network as SCL:
   #Tx[5].Start := (#Result < #SP.LL) AND #CMD.Start_A AND NOT #Use.Lim_Low;
   IF (#Result < #SP.LL) AND #CMD.Start_A AND NOT #Use.Lim_Low AND #Tx[5]."Exit" THEN
       #Alarms.%X5 := TRUE;
       #Alarm.LL := TRUE;
   END_IF;
END_REGION

REGION Network 18: Наличие любой ошибки
   RUNG wire#powerrail
      Contact( #Alarm.NC )
      wire#w1
      S_Coil( #CMD.Alarm )
   END_RUNG
   RUNG wire#powerrail
      Contact( #Alarm.SC )
   END_RUNG wire#w1
   RUNG wire#powerrail
      Contact( #Alarm.HH )
   END_RUNG wire#w1
   RUNG wire#powerrail
      Contact( #Alarm.LL )
   END_RUNG wire#w1
   RUNG wire#w1
      S_Coil( #S_Alarm )
   END_RUNG
   RUNG wire#w1
      S_Coil( "Alm_AI" )
   END_RUNG
   // the same network as SCL:
   IF #Alarm.NC OR #Alarm.SC OR #Alarm.HH OR #Alarm.LL THEN
       #CMD.Alarm := TRUE;
       #S_Alarm := TRUE;
       "Alm_AI" := TRUE;
   END_IF;
END_REGION

REGION Network 19: Сброс аварий
   RUNG wire#powerrail
      Contact( #CMD.Reset )
      Move(in := 2#0, out1 => #Alarms)
      wire#w1
      R_Coil( #Alarm.NC )
   END_RUNG
   RUNG wire#w1
      R_Coil( #Alarm.SC )
   END_RUNG
   RUNG wire#w1
      R_Coil( #Alarm.HH )
   END_RUNG
   RUNG wire#w1
      R_Coil( #Alarm.LL )
   END_RUNG
   RUNG wire#w1
      R_Coil( #CMD.Alarm )
   END_RUNG
   RUNG wire#w1
      R_Coil( #S_Alarm )
   END_RUNG
   // the same network as SCL:
   IF #CMD.Reset THEN
       #Alarms := 2#0;
       #Alarm.NC := FALSE;
       #Alarm.SC := FALSE;
       #Alarm.HH := FALSE;
       #Alarm.LL := FALSE;
       #CMD.Alarm := FALSE;
       #S_Alarm := FALSE;
   END_IF;
END_REGION

REGION Network 20: События датчика
   // 0 - датчик активирован
   // 1 - датчик деактивирован
   // 2 - датчик в ручном режиме
   // 3 - датчик в автоматическом режиме
   // 4 - сигнал ниже нижнего предупреждающего
   // 5 - сигнал в норме
   // 6 - сигнал выше верхнего предупреждающего
   // 7 - сигнал в норме
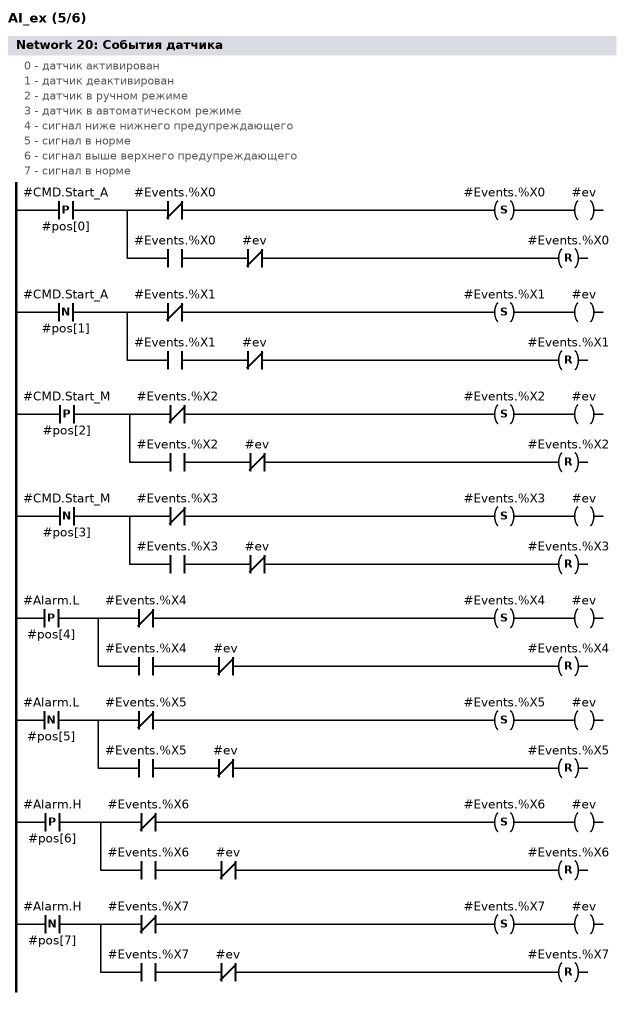
   RUNG wire#powerrail
      P_Contact(operand := #CMD.Start_A, bit := #pos[0])
      wire#w1
      I_Contact( #Events.%X0 )
      S_Coil( #Events.%X0 )
      Coil( #ev )
   END_RUNG
   RUNG wire#w1
      Contact( #Events.%X0 )
      I_Contact( #ev )
      R_Coil( #Events.%X0 )
   END_RUNG
   RUNG wire#powerrail
      N_Contact(operand := #CMD.Start_A, bit := #pos[1])
      wire#w2
      I_Contact( #Events.%X1 )
      S_Coil( #Events.%X1 )
      Coil( #ev )
   END_RUNG
   RUNG wire#w2
      Contact( #Events.%X1 )
      I_Contact( #ev )
      R_Coil( #Events.%X1 )
   END_RUNG
   RUNG wire#powerrail
      P_Contact(operand := #CMD.Start_M, bit := #pos[2])
      wire#w3
      I_Contact( #Events.%X2 )
      S_Coil( #Events.%X2 )
      Coil( #ev )
   END_RUNG
   RUNG wire#w3
      Contact( #Events.%X2 )
      I_Contact( #ev )
      R_Coil( #Events.%X2 )
   END_RUNG
   RUNG wire#powerrail
      N_Contact(operand := #CMD.Start_M, bit := #pos[3])
      wire#w4
      I_Contact( #Events.%X3 )
      S_Coil( #Events.%X3 )
      Coil( #ev )
   END_RUNG
   RUNG wire#w4
      Contact( #Events.%X3 )
      I_Contact( #ev )
      R_Coil( #Events.%X3 )
   END_RUNG
   RUNG wire#powerrail
      P_Contact(operand := #Alarm.L, bit := #pos[4])
      wire#w5
      I_Contact( #Events.%X4 )
      S_Coil( #Events.%X4 )
      Coil( #ev )
   END_RUNG
   RUNG wire#w5
      Contact( #Events.%X4 )
      I_Contact( #ev )
      R_Coil( #Events.%X4 )
   END_RUNG
   RUNG wire#powerrail
      N_Contact(operand := #Alarm.L, bit := #pos[5])
      wire#w6
      I_Contact( #Events.%X5 )
      S_Coil( #Events.%X5 )
      Coil( #ev )
   END_RUNG
   RUNG wire#w6
      Contact( #Events.%X5 )
      I_Contact( #ev )
      R_Coil( #Events.%X5 )
   END_RUNG
   RUNG wire#powerrail
      P_Contact(operand := #Alarm.H, bit := #pos[6])
      wire#w7
      I_Contact( #Events.%X6 )
      S_Coil( #Events.%X6 )
      Coil( #ev )
   END_RUNG
   RUNG wire#w7
      Contact( #Events.%X6 )
      I_Contact( #ev )
      R_Coil( #Events.%X6 )
   END_RUNG
   RUNG wire#powerrail
      N_Contact(operand := #Alarm.H, bit := #pos[7])
      wire#w8
      I_Contact( #Events.%X7 )
      S_Coil( #Events.%X7 )
      Coil( #ev )
   END_RUNG
   RUNG wire#w8
      Contact( #Events.%X7 )
      I_Contact( #ev )
      R_Coil( #Events.%X7 )
   END_RUNG
   // the same network as SCL:
   #_w1 := #CMD.Start_A AND NOT #pos[0];   // rising edge of #CMD.Start_A
   #pos[0] := #CMD.Start_A;
   #_w2 := #_w1 AND NOT #Events.%X0;
   IF #_w2 THEN #Events.%X0 := TRUE; END_IF;
   #ev := #_w2;
   IF #_w1 AND #Events.%X0 AND NOT #ev THEN #Events.%X0 := FALSE; END_IF;
   #_w3 := NOT #CMD.Start_A AND #pos[1];   // falling edge of #CMD.Start_A
   #pos[1] := #CMD.Start_A;
   #_w4 := #_w3 AND NOT #Events.%X1;
   IF #_w4 THEN #Events.%X1 := TRUE; END_IF;
   #ev := #_w4;
   IF #_w3 AND #Events.%X1 AND NOT #ev THEN #Events.%X1 := FALSE; END_IF;
   #_w5 := #CMD.Start_M AND NOT #pos[2];   // rising edge of #CMD.Start_M
   #pos[2] := #CMD.Start_M;
   #_w6 := #_w5 AND NOT #Events.%X2;
   IF #_w6 THEN #Events.%X2 := TRUE; END_IF;
   #ev := #_w6;
   IF #_w5 AND #Events.%X2 AND NOT #ev THEN #Events.%X2 := FALSE; END_IF;
   #_w7 := NOT #CMD.Start_M AND #pos[3];   // falling edge of #CMD.Start_M
   #pos[3] := #CMD.Start_M;
   #_w8 := #_w7 AND NOT #Events.%X3;
   IF #_w8 THEN #Events.%X3 := TRUE; END_IF;
   #ev := #_w8;
   IF #_w7 AND #Events.%X3 AND NOT #ev THEN #Events.%X3 := FALSE; END_IF;
   #_w9 := #Alarm.L AND NOT #pos[4];   // rising edge of #Alarm.L
   #pos[4] := #Alarm.L;
   #_w10 := #_w9 AND NOT #Events.%X4;
   IF #_w10 THEN #Events.%X4 := TRUE; END_IF;
   #ev := #_w10;
   IF #_w9 AND #Events.%X4 AND NOT #ev THEN #Events.%X4 := FALSE; END_IF;
   #_w11 := NOT #Alarm.L AND #pos[5];   // falling edge of #Alarm.L
   #pos[5] := #Alarm.L;
   #_w12 := #_w11 AND NOT #Events.%X5;
   IF #_w12 THEN #Events.%X5 := TRUE; END_IF;
   #ev := #_w12;
   IF #_w11 AND #Events.%X5 AND NOT #ev THEN #Events.%X5 := FALSE; END_IF;
   #_w13 := #Alarm.H AND NOT #pos[6];   // rising edge of #Alarm.H
   #pos[6] := #Alarm.H;
   #_w14 := #_w13 AND NOT #Events.%X6;
   IF #_w14 THEN #Events.%X6 := TRUE; END_IF;
   #ev := #_w14;
   IF #_w13 AND #Events.%X6 AND NOT #ev THEN #Events.%X6 := FALSE; END_IF;
   #_w15 := NOT #Alarm.H AND #pos[7];   // falling edge of #Alarm.H
   #pos[7] := #Alarm.H;
   #_w16 := #_w15 AND NOT #Events.%X7;
   IF #_w16 THEN #Events.%X7 := TRUE; END_IF;
   #ev := #_w16;
   IF #_w15 AND #Events.%X7 AND NOT #ev THEN #Events.%X7 := FALSE; END_IF;
END_REGION

REGION Network 21: Статус входа
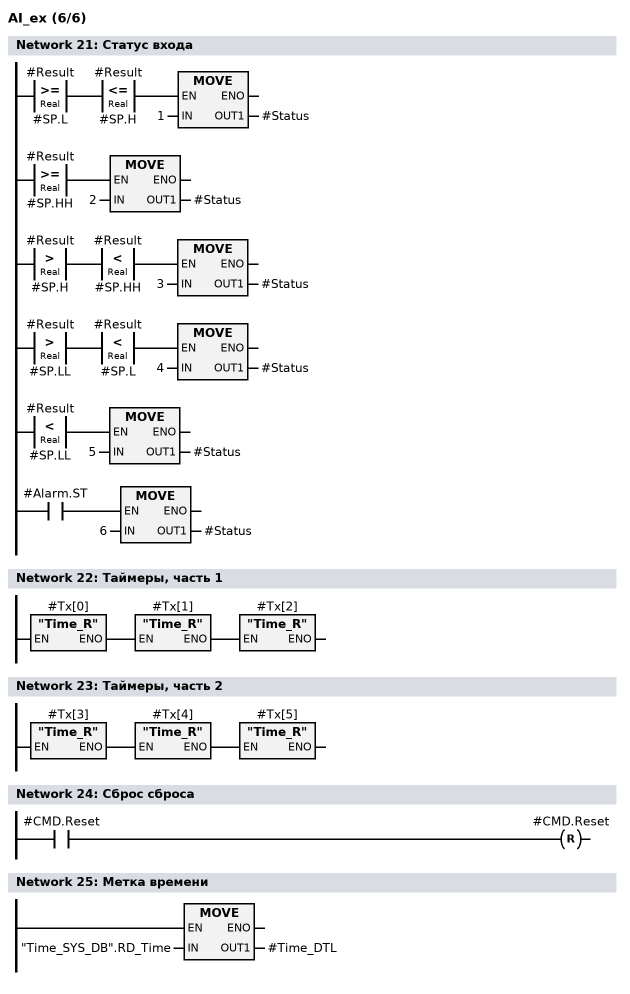
   RUNG wire#powerrail
      { S7_Templates := "SrcType := Real" } GE_Contact(in1 := #Result, in2 := #SP.L)
      { S7_Templates := "SrcType := Real" } LE_Contact(in1 := #Result, in2 := #SP.H)
      Move(in := 1, out1 => #Status)
   END_RUNG
   RUNG wire#powerrail
      { S7_Templates := "SrcType := Real" } GE_Contact(in1 := #Result, in2 := #SP.HH)
      Move(in := 2, out1 => #Status)
   END_RUNG
   RUNG wire#powerrail
      { S7_Templates := "SrcType := Real" } GT_Contact(in1 := #Result, in2 := #SP.H)
      { S7_Templates := "SrcType := Real" } LT_Contact(in1 := #Result, in2 := #SP.HH)
      Move(in := 3, out1 => #Status)
   END_RUNG
   RUNG wire#powerrail
      { S7_Templates := "SrcType := Real" } GT_Contact(in1 := #Result, in2 := #SP.LL)
      { S7_Templates := "SrcType := Real" } LT_Contact(in1 := #Result, in2 := #SP.L)
      Move(in := 4, out1 => #Status)
   END_RUNG
   RUNG wire#powerrail
      { S7_Templates := "SrcType := Real" } LT_Contact(in1 := #Result, in2 := #SP.LL)
      Move(in := 5, out1 => #Status)
   END_RUNG
   RUNG wire#powerrail
      Contact( #Alarm.ST )
      Move(in := 6, out1 => #Status)
   END_RUNG
   // the same network as SCL:
   IF (#Result >= #SP.L) AND (#Result <= #SP.H) THEN #Status := 1; END_IF;
   IF #Result >= #SP.HH THEN #Status := 2; END_IF;
   IF (#Result > #SP.H) AND (#Result < #SP.HH) THEN #Status := 3; END_IF;
   IF (#Result > #SP.LL) AND (#Result < #SP.L) THEN #Status := 4; END_IF;
   IF #Result < #SP.LL THEN #Status := 5; END_IF;
   IF #Alarm.ST THEN #Status := 6; END_IF;
END_REGION

REGION Network 22: Таймеры, часть 1
   RUNG wire#powerrail
      #Tx[0]()
      #Tx[1]()
      #Tx[2]()
   END_RUNG
   // the same network as SCL:
   #Tx[0](ENO => #_w1);   // "Time_R"
   #Tx[1](EN := #_w1, ENO => #_w2);   // "Time_R"
   IF #_w2 THEN
       #Tx[2]();   // "Time_R"
   END_IF;
END_REGION

REGION Network 23: Таймеры, часть 2
   RUNG wire#powerrail
      #Tx[3]()
      #Tx[4]()
      #Tx[5]()
   END_RUNG
   // the same network as SCL:
   #Tx[3](ENO => #_w1);   // "Time_R"
   #Tx[4](EN := #_w1, ENO => #_w2);   // "Time_R"
   IF #_w2 THEN
       #Tx[5]();   // "Time_R"
   END_IF;
END_REGION

REGION Network 24: Сброс сброса
   RUNG wire#powerrail
      Contact( #CMD.Reset )
      R_Coil( #CMD.Reset )
   END_RUNG
   // the same network as SCL:
   IF #CMD.Reset THEN #CMD.Reset := FALSE; END_IF;
END_REGION

REGION Network 25: Метка времени
   RUNG wire#powerrail
      Move(in := "Time_SYS_DB".RD_Time, out1 => #Time_DTL)
   END_RUNG
   // the same network as SCL:
   #Time_DTL := "Time_SYS_DB".RD_Time;
END_REGION
END_FUNCTION_BLOCK

FUNCTION "drv_Mode" : Void   // FC150, LAD
{ S7_Optimized_Access := 'FALSE' }
VERSION : 0.1
// stored: AutoNumber false, IsIECCheckEnabled false, SetENOAutomatically false, UDAEnableTagReadback false
   VAR_INPUT
      CMD : "CMD";   // Основные команды / Блок команд
      All_Block : Bool;   // Аварийная блокировка
   END_VAR
   VAR_OUTPUT
      Mode : Int;   // Режим работы
   END_VAR
BEGIN

REGION Network 1: Автоматический режим
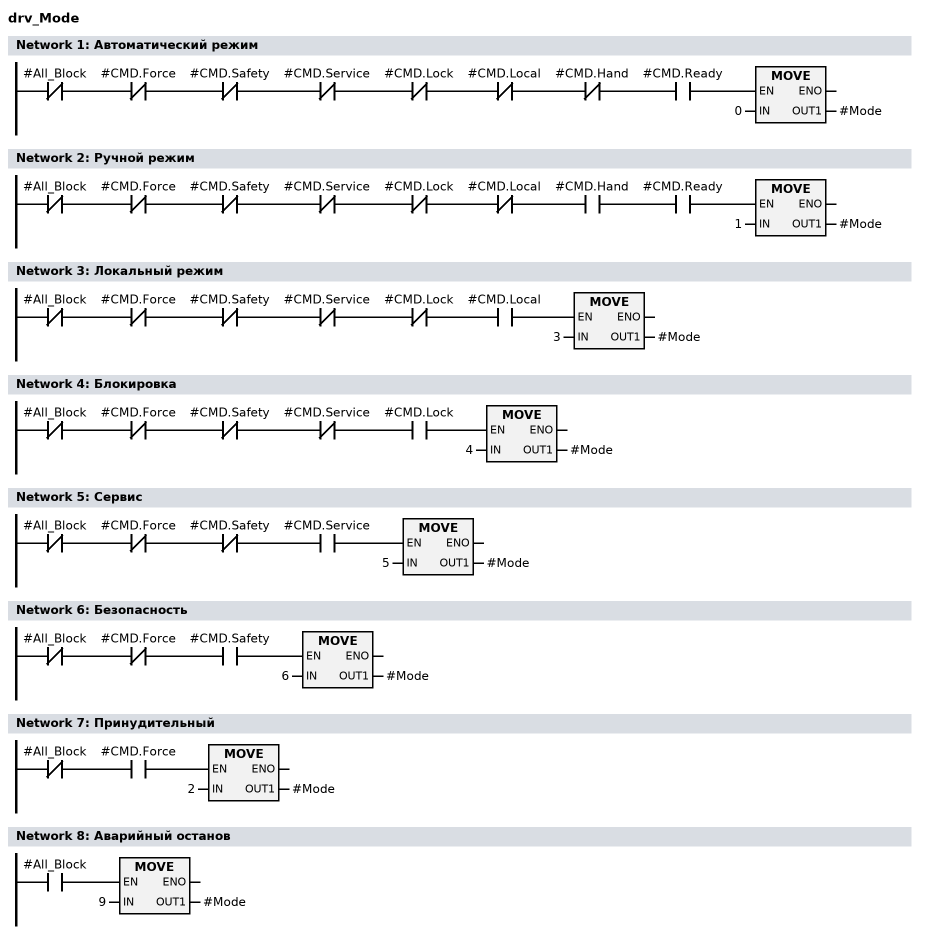
   RUNG wire#powerrail
      I_Contact( #All_Block )
      I_Contact( #CMD.Force )
      I_Contact( #CMD.Safety )
      I_Contact( #CMD.Service )
      I_Contact( #CMD.Lock )
      I_Contact( #CMD.Local )
      I_Contact( #CMD.Hand )
      Contact( #CMD.Ready )
      { S7_GenerateENO := "TRUE" } Move(in := 0, out1 => #Mode)
   END_RUNG
   // the same network as SCL:
   IF NOT #All_Block AND NOT #CMD.Force AND NOT #CMD.Safety AND NOT #CMD.Service AND NOT #CMD.Lock AND NOT #CMD.Local AND NOT #CMD.Hand AND #CMD.Ready THEN
       #Mode := 0;
   END_IF;
END_REGION

REGION Network 2: Ручной режим
   RUNG wire#powerrail
      I_Contact( #All_Block )
      I_Contact( #CMD.Force )
      I_Contact( #CMD.Safety )
      I_Contact( #CMD.Service )
      I_Contact( #CMD.Lock )
      I_Contact( #CMD.Local )
      Contact( #CMD.Hand )
      Contact( #CMD.Ready )
      { S7_GenerateENO := "TRUE" } Move(in := 1, out1 => #Mode)
   END_RUNG
   // the same network as SCL:
   IF NOT #All_Block AND NOT #CMD.Force AND NOT #CMD.Safety AND NOT #CMD.Service AND NOT #CMD.Lock AND NOT #CMD.Local AND #CMD.Hand AND #CMD.Ready THEN
       #Mode := 1;
   END_IF;
END_REGION

REGION Network 3: Локальный режим
   RUNG wire#powerrail
      I_Contact( #All_Block )
      I_Contact( #CMD.Force )
      I_Contact( #CMD.Safety )
      I_Contact( #CMD.Service )
      I_Contact( #CMD.Lock )
      Contact( #CMD.Local )
      { S7_GenerateENO := "TRUE" } Move(in := 3, out1 => #Mode)
   END_RUNG
   // the same network as SCL:
   IF NOT #All_Block AND NOT #CMD.Force AND NOT #CMD.Safety AND NOT #CMD.Service AND NOT #CMD.Lock AND #CMD.Local THEN
       #Mode := 3;
   END_IF;
END_REGION

REGION Network 4: Блокировка
   RUNG wire#powerrail
      I_Contact( #All_Block )
      I_Contact( #CMD.Force )
      I_Contact( #CMD.Safety )
      I_Contact( #CMD.Service )
      Contact( #CMD.Lock )
      { S7_GenerateENO := "TRUE" } Move(in := 4, out1 => #Mode)
   END_RUNG
   // the same network as SCL:
   IF NOT #All_Block AND NOT #CMD.Force AND NOT #CMD.Safety AND NOT #CMD.Service AND #CMD.Lock THEN
       #Mode := 4;
   END_IF;
END_REGION

REGION Network 5: Сервис
   RUNG wire#powerrail
      I_Contact( #All_Block )
      I_Contact( #CMD.Force )
      I_Contact( #CMD.Safety )
      Contact( #CMD.Service )
      { S7_GenerateENO := "TRUE" } Move(in := 5, out1 => #Mode)
   END_RUNG
   // the same network as SCL:
   IF NOT #All_Block AND NOT #CMD.Force AND NOT #CMD.Safety AND #CMD.Service THEN #Mode := 5; END_IF;
END_REGION

REGION Network 6: Безопасность
   RUNG wire#powerrail
      I_Contact( #All_Block )
      I_Contact( #CMD.Force )
      Contact( #CMD.Safety )
      { S7_GenerateENO := "TRUE" } Move(in := 6, out1 => #Mode)
   END_RUNG
   // the same network as SCL:
   IF NOT #All_Block AND NOT #CMD.Force AND #CMD.Safety THEN #Mode := 6; END_IF;
END_REGION

REGION Network 7: Принудительный
   RUNG wire#powerrail
      I_Contact( #All_Block )
      Contact( #CMD.Force )
      { S7_GenerateENO := "TRUE" } Move(in := 2, out1 => #Mode)
   END_RUNG
   // the same network as SCL:
   IF NOT #All_Block AND #CMD.Force THEN #Mode := 2; END_IF;
END_REGION

REGION Network 8: Аварийный останов
   RUNG wire#powerrail
      Contact( #All_Block )
      { S7_GenerateENO := "TRUE" } Move(in := 9, out1 => #Mode)
   END_RUNG
   // the same network as SCL:
   IF #All_Block THEN #Mode := 9; END_IF;
END_REGION
END_FUNCTION

FUNCTION_BLOCK "Converter_LAD"   // FB98, LAD
{ S7_Optimized_Access := 'FALSE' }
VERSION : 0.1
// stored: AutoNumber false, IsIECCheckEnabled false, SetENOAutomatically false, UDAEnableTagReadback false
   VAR_INPUT
      Signal : Real;   // Входной сигнал
   END_VAR
   VAR_OUTPUT
      Result : Real;   // Результат линеаризации
   END_VAR
   VAR DB_SPECIFIC
      Use_Min_In { S7_SetPoint := 'True'} : Bool;   // Отсекать входные значения ниже минимума
      Use_Max_In { S7_SetPoint := 'True'} : Bool;   // Отсекать входные значения выше максимума
      Use_Min_Out { S7_SetPoint := 'True'} : Bool;   // Отсекать результат ниже минимума
      Use_Max_Out { S7_SetPoint := 'True'} : Bool;   // Отсекать результат выше максимума
      IO { S7_SetPoint := 'True'} : Bool;   // Входной/Выходной режим
      Inverse { S7_SetPoint := 'True'} : Bool;   // Инверсия выхода
      Min_In { S7_SetPoint := 'True'} : Real;   // Минимальный входной сигнал
      Min_Out { S7_SetPoint := 'True'} : Real;   // Минимальный выходной сигнал
      Max_In { S7_SetPoint := 'True'} : Real;   // Максимальный входной сигнал
      Max_Out { S7_SetPoint := 'True'} : Real;   // Максимальный выходной сигнал
   END_VAR
   VAR_TEMP
      Range_In : Real;   // Диапазон входного сигнала
      Range_Out : Real;   // Диапазон выходного сигнала
      T_T : Real;   // Соотношение диапазонов
      R_Sig : Real;   // Поправка на отрицательные значения
   END_VAR
BEGIN

REGION Network 1: Проверка нижнего уровня входного сигнала
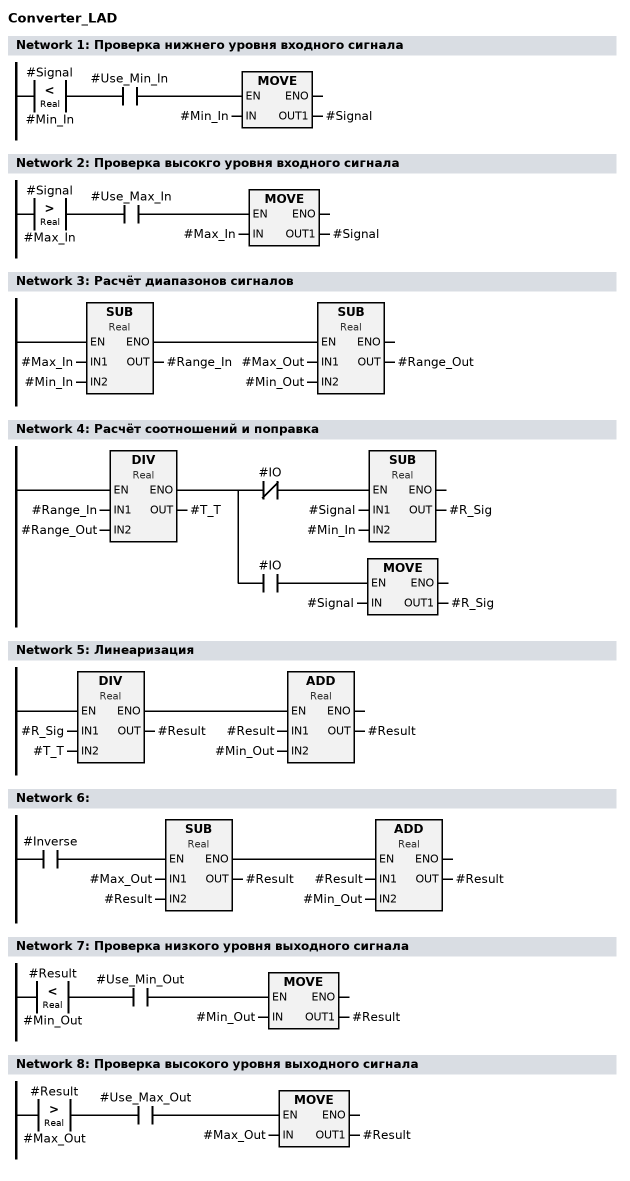
   RUNG wire#powerrail
      { S7_Templates := "SrcType := Real" } LT_Contact(in1 := #Signal, in2 := #Min_In)
      Contact( #Use_Min_In )
      { S7_GenerateENO := "TRUE" } Move(in := #Min_In, out1 => #Signal)
   END_RUNG
   // the same network as SCL:
   IF (#Signal < #Min_In) AND #Use_Min_In THEN #Signal := #Min_In; END_IF;
END_REGION

REGION Network 2: Проверка высокго уровня входного сигнала
   RUNG wire#powerrail
      { S7_Templates := "SrcType := Real" } GT_Contact(in1 := #Signal, in2 := #Max_In)
      Contact( #Use_Max_In )
      { S7_GenerateENO := "TRUE" } Move(in := #Max_In, out1 => #Signal)
   END_RUNG
   // the same network as SCL:
   IF (#Signal > #Max_In) AND #Use_Max_In THEN #Signal := #Max_In; END_IF;
END_REGION

REGION Network 3: Расчёт диапазонов сигналов
   RUNG wire#powerrail
      { S7_Templates := "SrcType := Real"; S7_GenerateENO := "TRUE" } Sub(in1 := #Max_In, in2 := #Min_In, out => #Range_In)
      { S7_Templates := "SrcType := Real"; S7_GenerateENO := "TRUE" } Sub(in1 := #Max_Out, in2 := #Min_Out, out => #Range_Out)
   END_RUNG
   // the same network as SCL:
   // ENO of a box is taken as its EN; it also drops when the box reports an error
   #Range_In := #Max_In - #Min_In;
   #Range_Out := #Max_Out - #Min_Out;
END_REGION

REGION Network 4: Расчёт соотношений и поправка
   RUNG wire#powerrail
      { S7_Templates := "SrcType := Real"; S7_GenerateENO := "TRUE" } Div(in1 := #Range_In, in2 := #Range_Out, out => #T_T)
      wire#w1
      I_Contact( #IO )
      { S7_Templates := "SrcType := Real"; S7_GenerateENO := "TRUE" } Sub(in1 := #Signal, in2 := #Min_In, out => #R_Sig)
   END_RUNG
   RUNG wire#w1
      Contact( #IO )
      { S7_GenerateENO := "TRUE" } Move(in := #Signal, out1 => #R_Sig)
   END_RUNG
   // the same network as SCL:
   // ENO of a box is taken as its EN; it also drops when the box reports an error
   #T_T := #Range_In / #Range_Out;
   IF NOT #IO THEN #R_Sig := #Signal - #Min_In; END_IF;
   IF #IO THEN #R_Sig := #Signal; END_IF;
END_REGION

REGION Network 5: Линеаризация
   RUNG wire#powerrail
      { S7_Templates := "SrcType := Real"; S7_GenerateENO := "TRUE" } Div(in1 := #R_Sig, in2 := #T_T, out => #Result)
      { S7_Templates := "SrcType := Real"; S7_GenerateENO := "TRUE" } Add(in1 := #Result, in2 := #Min_Out, out => #Result)
   END_RUNG
   // the same network as SCL:
   // ENO of a box is taken as its EN; it also drops when the box reports an error
   #Result := #R_Sig / #T_T;
   #Result := #Result + #Min_Out;
END_REGION

REGION Network 6
   RUNG wire#powerrail
      Contact( #Inverse )
      { S7_Templates := "SrcType := Real"; S7_GenerateENO := "TRUE" } Sub(in1 := #Max_Out, in2 := #Result, out => #Result)
      { S7_Templates := "SrcType := Real"; S7_GenerateENO := "TRUE" } Add(in1 := #Result, in2 := #Min_Out, out => #Result)
   END_RUNG
   // the same network as SCL:
   // ENO of a box is taken as its EN; it also drops when the box reports an error
   IF #Inverse THEN
       #Result := #Max_Out - #Result;
       #Result := #Result + #Min_Out;
   END_IF;
END_REGION

REGION Network 7: Проверка низкого уровня выходного сигнала
   RUNG wire#powerrail
      { S7_Templates := "SrcType := Real" } LT_Contact(in1 := #Result, in2 := #Min_Out)
      Contact( #Use_Min_Out )
      { S7_GenerateENO := "TRUE" } Move(in := #Min_Out, out1 => #Result)
   END_RUNG
   // the same network as SCL:
   IF (#Result < #Min_Out) AND #Use_Min_Out THEN #Result := #Min_Out; END_IF;
END_REGION

REGION Network 8: Проверка высокого уровня выходного сигнала
   RUNG wire#powerrail
      { S7_Templates := "SrcType := Real" } GT_Contact(in1 := #Result, in2 := #Max_Out)
      Contact( #Use_Max_Out )
      { S7_GenerateENO := "TRUE" } Move(in := #Max_Out, out1 => #Result)
   END_RUNG
   // the same network as SCL:
   IF (#Result > #Max_Out) AND #Use_Max_Out THEN #Result := #Max_Out; END_IF;
END_REGION
END_FUNCTION_BLOCK

FUNCTION_BLOCK "Time_R"   // FB91, LAD
{ S7_Optimized_Access := 'FALSE' }
VERSION : 0.1
// stored: AutoNumber false, IsIECCheckEnabled false, SetENOAutomatically false, UDAEnableTagReadback false
   VAR DB_SPECIFIC
      SP { S7_SetPoint := 'True'} : Real := 1.0;   // Уставка
      Now : Real;   // Текущий счёт
      One { S7_SetPoint := 'True'} : Real := 0.1;   // Вес импульса
      Progress : Real;   // Прогресс выполнения
      Start : Bool;   // Запуск
      "Exit" : Bool;   // Счёт завершён
      Pause : Bool;   // Пауза
      Reset : Bool;   // Сброс счёта
   END_VAR
   VAR_TEMP   // added for the SCL form of the ladder/FBD networks
      _w1 : Bool;
   END_VAR
BEGIN

REGION Network 1: Подсчёт времени
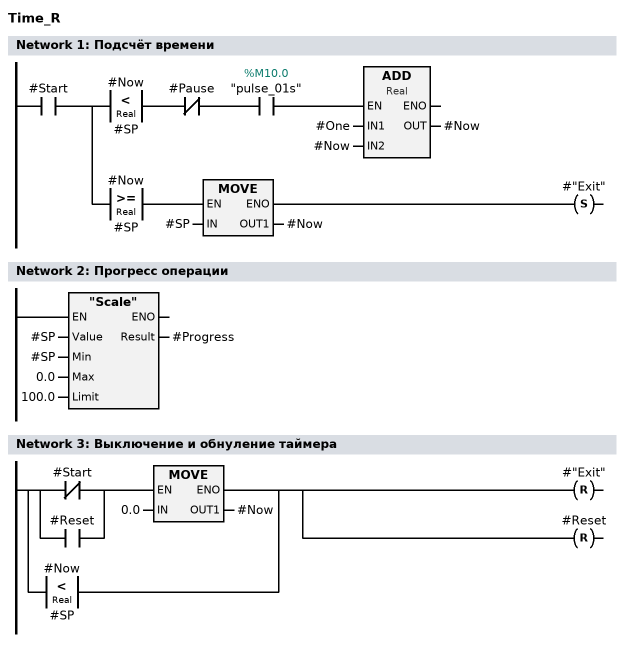
   RUNG wire#powerrail
      Contact( #Start )
      wire#w1
      { S7_Templates := "SrcType := Real" } LT_Contact(in1 := #Now, in2 := #SP)
      I_Contact( #Pause )
      Contact( "pulse_01s" )
      { S7_Templates := "SrcType := Real"; S7_GenerateENO := "TRUE" } Add(in1 := #One, in2 := #Now, out => #Now)
   END_RUNG
   RUNG wire#w1
      { S7_Templates := "SrcType := Real" } GE_Contact(in1 := #Now, in2 := #SP)
      Move(in := #SP, out1 => #Now)
      S_Coil( #"Exit" )
   END_RUNG
   // the same network as SCL:
   IF #Start AND (#Now < #SP) AND NOT #Pause AND "pulse_01s" THEN #Now := #One + #Now; END_IF;
   #_w1 := #Start AND (#Now >= #SP);
   IF #_w1 THEN
       #Now := #SP;
       #"Exit" := TRUE;
   END_IF;
END_REGION

REGION Network 2: Прогресс операции
   RUNG wire#powerrail
      "Scale"(Value := #SP, Min := #SP, Max := 0.0, Limit := 100.0, Result => #Progress)
   END_RUNG
   // the same network as SCL:
   "Scale"(Value := #SP, Min := #SP, Max := 0.0, Limit := 100.0, Result => #Progress);
END_REGION

REGION Network 3: Выключение и обнуление таймера
   RUNG wire#powerrail
      I_Contact( #Start )
      wire#w1
      { S7_GenerateENO := "TRUE" } Move(in := 0.0, out1 => #Now)
      wire#w2
      R_Coil( #"Exit" )
   END_RUNG
   RUNG wire#powerrail
      Contact( #Reset )
   END_RUNG wire#w1
   RUNG wire#powerrail
      { S7_Templates := "SrcType := Real" } LT_Contact(in1 := #Now, in2 := #SP)
   END_RUNG wire#w2
   RUNG wire#w2
      R_Coil( #Reset )
   END_RUNG
   // the same network as SCL:
   // ENO of a box is taken as its EN; it also drops when the box reports an error
   #_w1 := NOT #Start OR #Reset;
   IF #_w1 THEN #Now := 0.0; END_IF;
   IF #_w1 OR (#Now < #SP) THEN
       #"Exit" := FALSE;
       #Reset := FALSE;
   END_IF;
END_REGION
END_FUNCTION_BLOCK

FUNCTION_BLOCK "ModBus"
{ S7_Optimized_Access := 'TRUE' }
VERSION : 0.1
   VAR 
      Step : Int;   // Шаг опроса
      "type" : Int;   // тип устройства
      type_max : Int := 1;   // общее кол-во типов устройства
      cnt : Int;   // номер опрашиваемого устройства
      cnt_max : Int := 10;   // общее количество устройств
      CMD : Struct
         DIS : Bool;
         REQ : Bool;
         BUSY : Bool;
         DONE : Bool;
         ERROR : Bool;
         STATUS : Word;
      END_STRUCT;
      CFG : Struct
         ADDR : UInt;
         Register : UDInt;
         Length : UInt;
         IP {InstructionName := 'IP_V4'; LibVersion := '1.0'; S7_SetPoint := 'False'} : IP_V4;
         Port { S7_SetPoint := 'True'} : UInt;
         Mode : USInt;
      END_STRUCT;
      Clock { S7_SetPoint := 'False'} : Array[0..10] of "Time_S";
      test : Int;
      test_run : Bool;
   END_VAR

   VAR_TEMP 
      fc_read : Bool;
      fc_write : Bool;
      x : Int;
   END_VAR


BEGIN
	// Общее количество устройств для опроса
	IF #cnt > #cnt_max THEN
	    #cnt := 0;
	END_IF;
	//#cnt := 3;
	//  Цикл опроса
	CASE #Step OF
	    0:  //  Шаг 0 - параметры подключения
	        #Step := 1;
	
	                #CFG.IP := "tGw_DB".tGw["FE_DB".FE[#cnt].ID].IP;
	                #CFG."Port" := "tGw_DB".tGw["FE_DB".FE[#cnt].ID]."Port";
	                #CFG.ADDR := "FE_DB".FE["FE_DB".FE[#cnt].ID].ADDR;
	
	        IF NOT "ModBus_TCP_DB".CONNECT.ActiveEstablished THEN
	            #Step := 10;
	        END_IF;
	    1:  //  Шаг 1 - параметры чтения
	
	        #CFG.Register := 0;
	        #CFG.Length := 12;
	        #CFG.Mode := 104;
	
	        IF NOT #CMD.BUSY AND NOT #CMD.DONE THEN
	            #Step := 2;
	            //#CMD.DIS := FALSE;
	        END_IF;
	    2:  // Шаг 2 - чтение данных
	        #CMD.REQ := TRUE;
	        #Clock[0].Start := TRUE;
	        //успешное чтение данных
	        IF #CMD.DONE THEN
	            %DB5.DBW42 := %DB40.DBW0;
	            %DB5.DBW44 := %DB40.DBW2;
	            %DB5.DBW46 := %DB40.DBW4;
	            %DB5.DBW48 := %DB40.DBW6;
	            %DB5.DBW50 := %DB40.DBW8;
	            %DB5.DBW52 := %DB40.DBW10;
	            %DB5.DBW54 := %DB40.DBW12;
	            %DB5.DBW56 := %DB40.DBW14;
	            %DB5.DBW58 := %DB40.DBW16;
	            %DB5.DBW60 := %DB40.DBW18;
	            %DB5.DBW62 := %DB40.DBW20;
	            %DB5.DBW64 := %DB40.DBW22;
	            "FE_DB".FE[1].Flow := "FE_DB".FE[1].Flow * 3600;
	                    "FE_DB".FE[#cnt].Link := TRUE;
	                    #Step := 10;
	        END_IF;
	        //ошибка при чтении
	        IF #CMD.ERROR OR #Clock[0]."Exit" THEN
	
	                    "FE_DB".FE[#cnt].Link := FALSE;
	                    "FE_DB".FE[#cnt].NoRead := TRUE;
	                    #Step := 10;
	
	        END_IF;
	    10: //  Шаг 10 - конец опроса
	        #CMD.REQ := FALSE;
	        //#CMD.DIS := TRUE;
	        #cnt := 1;
	        //сброс таймеров
	        FOR #x := 0 TO 10 BY 1 DO
	            #Clock[#x].Start := FALSE;
	        END_FOR;
	        //очистка буфера
	        FOR #x := 0 TO 20 BY 1 DO
	            "ModBus_TCP_DB".DATA[#x] := 0;
	        END_FOR;
	        //конец цикла
	        #Step := 0;
	END_CASE;
	
	//вызов таймеров на исполнение
	FOR #x := 0 TO 10 BY 1 DO
	    #Clock[#x]();
	END_FOR;
	
	        
END_FUNCTION_BLOCK

FUNCTION_BLOCK "Time_S"   // FB90, LAD
{ S7_Optimized_Access := 'FALSE' }
VERSION : 0.1
// stored: AutoNumber false, IsIECCheckEnabled false, SetENOAutomatically false, UDAEnableTagReadback false
   VAR DB_SPECIFIC
      SP { S7_SetPoint := 'True'} : Int := 2;   // Уставка
      Now : Int;   // Текущий счёт
      Start : Bool;   // Запуск
      "Exit" : Bool;   // Счёт завершён
      Pause : Bool;   // Пауза
      Reset : Bool;   // Сброс таймера
   END_VAR
   VAR_TEMP   // added for the SCL form of the ladder/FBD networks
      _w1 : Bool;
   END_VAR
BEGIN

REGION Network 1: Подсчёт времени
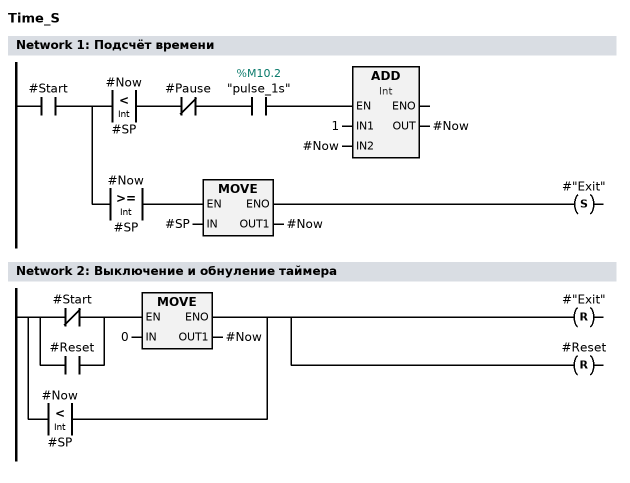
   RUNG wire#powerrail
      Contact( #Start )
      wire#w1
      { S7_Templates := "SrcType := Int" } LT_Contact(in1 := #Now, in2 := #SP)
      I_Contact( #Pause )
      Contact( "pulse_1s" )
      { S7_Templates := "SrcType := Int"; S7_GenerateENO := "TRUE" } Add(in1 := 1, in2 := #Now, out => #Now)
   END_RUNG
   RUNG wire#w1
      { S7_Templates := "SrcType := Int" } GE_Contact(in1 := #Now, in2 := #SP)
      { S7_GenerateENO := "TRUE" } Move(in := #SP, out1 => #Now)
      S_Coil( #"Exit" )
   END_RUNG
   // the same network as SCL:
   // ENO of a box is taken as its EN; it also drops when the box reports an error
   IF #Start AND (#Now < #SP) AND NOT #Pause AND "pulse_1s" THEN #Now := 1 + #Now; END_IF;
   #_w1 := #Start AND (#Now >= #SP);
   IF #_w1 THEN
       #Now := #SP;
       #"Exit" := TRUE;
   END_IF;
END_REGION

REGION Network 2: Выключение и обнуление таймера
   RUNG wire#powerrail
      I_Contact( #Start )
      wire#w1
      { S7_GenerateENO := "TRUE" } Move(in := 0, out1 => #Now)
      wire#w2
      R_Coil( #"Exit" )
   END_RUNG
   RUNG wire#powerrail
      Contact( #Reset )
   END_RUNG wire#w1
   RUNG wire#powerrail
      { S7_Templates := "SrcType := Int" } LT_Contact(in1 := #Now, in2 := #SP)
   END_RUNG wire#w2
   RUNG wire#w2
      R_Coil( #Reset )
   END_RUNG
   // the same network as SCL:
   // ENO of a box is taken as its EN; it also drops when the box reports an error
   #_w1 := NOT #Start OR #Reset;
   IF #_w1 THEN #Now := 0; END_IF;
   IF #_w1 OR (#Now < #SP) THEN
       #"Exit" := FALSE;
       #Reset := FALSE;
   END_IF;
END_REGION
END_FUNCTION_BLOCK

FUNCTION_BLOCK "ModBus_TCP"   // FB40, LAD
TITLE = Блок опроса ModBus TCP
{ S7_Optimized_Access := 'FALSE' }
VERSION : 0.1
// ВНИМАНИЕ!  Через один аппаратный порт контроллера можно проводить множество различных опросов по ModBus TCP. Для этого у каждого экземпляра должен быть указан уникальный CONNECT.ID.
// 
// Для каждого уникального CONNECT.ID / внешней ветки / точки подключения (IP, RemotePort) рекомендуется использовать отдельный экземпляр функционального блока. Например, при использовании tGW-735 имеющего 3 порта подключения с RemotePort = 502, 503 и 504 соответственно (но общий IP адрес) рекомендуется использовать три отдельных блока ModBus_TCP с уникальными CONNECT.ID.
// 
// Каждая точка чтения/записи = 1 экземпляр DEV_Config, количество элементов в массиве можно менять по необходимости, итоговое количество элементов массива указывается в теге Limit.
// 
// Для режима чтения необходимо указать:
// - MODE = 0
// - Source_DB = 40 (номер DB Modbus_TCP_DB)
// - SourceOFFSET = 0
// - Target_DB = xx (номер DB, куда необходимо положить прочитанные данные)
// - Target_OFFSET = xx (номер байта, начиная с которого кладутся прочитанные данные в выбранный DB)
// 
// Для режима опроса необходимо указать:
// - MODE = 1
// - Source_DB = xx (номер DB, откуда необходимо взять данные для передачи)
// - Source_OFFSET = xx (номер байта, начиная с которого берутся данные для передачи)
// - Target_DB = 40 (номер DB Modbus_TCP_DB)
// - Target_OFFSET = 0
// stored: AutoNumber false, IsIECCheckEnabled false, SetENOAutomatically false, UDAEnableTagReadback false
   VAR DB_SPECIFIC
      DATA : Array[0..100] of Word;   // Массив данных
      CONNECT { S7_SetPoint := 'True'} : TCON_IP_v4;
   END_VAR
   // CONNECT.InterfaceId := 64;
   // CONNECT.ID := 16#0001;
   // CONNECT.ConnectionType := 16#0B;
   // CONNECT.ActiveEstablished := TRUE;
   // CONNECT.RemoteAddress.ADDR[1] := 16#C0;
   // CONNECT.RemoteAddress.ADDR[2] := 16#A8;
   // CONNECT.RemoteAddress.ADDR[3] := 16#00;
   // CONNECT.RemoteAddress.ADDR[4] := 16#0A;
   // CONNECT.RemotePort := 502;
   // CONNECT.LocalPort := 0;
BEGIN

REGION Network 1
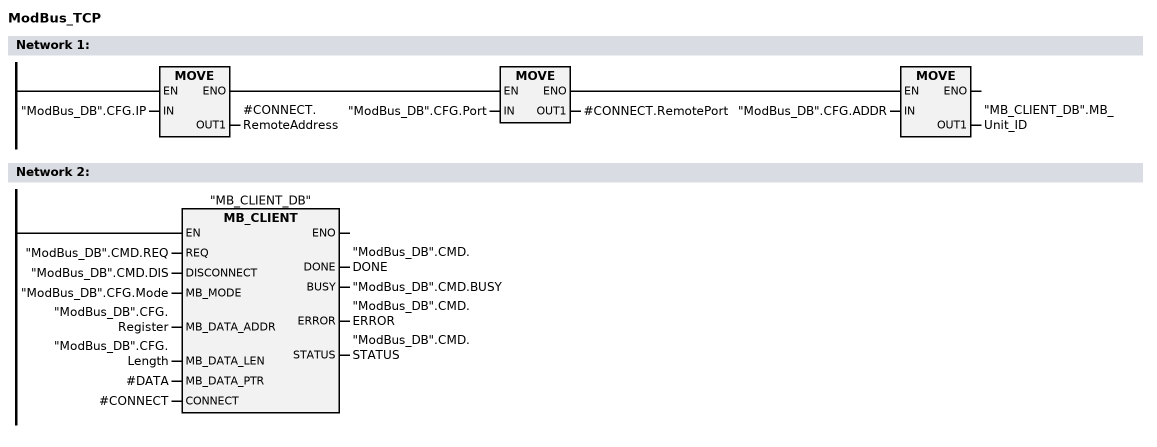
   RUNG wire#powerrail
      Move(in := "ModBus_DB".CFG.IP, out1 => #CONNECT.RemoteAddress)
      Move(in := "ModBus_DB".CFG.Port, out1 => #CONNECT.RemotePort)
      Move(in := "ModBus_DB".CFG.ADDR, out1 => "MB_CLIENT_DB".MB_Unit_ID)
   END_RUNG
   // the same network as SCL:
   #CONNECT.RemoteAddress := "ModBus_DB".CFG.IP;
   #CONNECT.RemotePort := "ModBus_DB".CFG.Port;
   "MB_CLIENT_DB".MB_Unit_ID := "ModBus_DB".CFG.ADDR;
END_REGION

REGION Network 2
   RUNG wire#powerrail
      "MB_CLIENT_DB".MB_CLIENT(REQ := "ModBus_DB".CMD.REQ, DISCONNECT := "ModBus_DB".CMD.DIS, MB_MODE := "ModBus_DB".CFG.Mode, MB_DATA_ADDR := "ModBus_DB".CFG.Register, MB_DATA_LEN := "ModBus_DB".CFG.Length, MB_DATA_PTR := #DATA, CONNECT := #CONNECT, DONE => "ModBus_DB".CMD.DONE, BUSY => "ModBus_DB".CMD.BUSY, ERROR => "ModBus_DB".CMD.ERROR, STATUS => "ModBus_DB".CMD.STATUS)
   END_RUNG
   // the same network as SCL:
   "MB_CLIENT_DB"(REQ := "ModBus_DB".CMD.REQ,   // MB_CLIENT
                  DISCONNECT := "ModBus_DB".CMD.DIS,
                  MB_MODE := "ModBus_DB".CFG.Mode,
                  MB_DATA_ADDR := "ModBus_DB".CFG.Register,
                  MB_DATA_LEN := "ModBus_DB".CFG.Length,
                  MB_DATA_PTR := #DATA,
                  CONNECT := #CONNECT,
                  DONE => "ModBus_DB".CMD.DONE,
                  BUSY => "ModBus_DB".CMD.BUSY,
                  ERROR => "ModBus_DB".CMD.ERROR,
                  STATUS => "ModBus_DB".CMD.STATUS);
END_REGION
END_FUNCTION_BLOCK

FUNCTION_BLOCK "Comm_SKD1"
{ S7_Optimized_Access := 'FALSE' }
VERSION : 0.1
   VAR 
      From_SKD1 : Struct
         watchdog : Int;
         LE_1 : Int;
         LE_2 : Int;
         LE_3 : Int;
         LE_4 : Int;
         SP_FE : Int;
         SP_M : Int;
         CMD : Struct
            REQ : Bool;
            Reset : Bool;
            Hand : Bool;
            Start_M : Bool;
         END_STRUCT;
         Valves : Struct
            ID : Int;
            Local : Array[0..15] of Bool;
            Mode : Array[1..10] of Int;
            Status : Array[1..10] of Int;
         END_STRUCT;
      END_STRUCT;
      To_SKD1 : Struct
         watchdog : Int;
         LE_SKV : Int;
         res_h : DInt;
         LE : Int;
         TE : Int;
         PE_1 : Int;
         PE_2 : Int;
         PE_3 : Int;
         PE_4 : Int;
         FE : Int;
         C : Int;
         Status : Int;
         STATE : Struct
            Ready : Bool;
            Local : Bool;
            Warning : Bool;
            Alarm : Bool;
            LS : Bool;
            Lock : Bool;
         END_STRUCT;
         Valves : Struct
            ID : Int;
            REQ : Array[0..15] of Bool;
         END_STRUCT;
      END_STRUCT;
      Alarm : Struct
         Link : Bool;
      END_STRUCT;
      watchdog_control : Int;
      ID : Int;
      LE_1 : Real;
      LE_2 : Real;
      LE_3 : Real;
      LE_4 : Real;
      Valve_Name { S7_SetPoint := 'True'} : Array[1..10] of String[4];
      Clock { S7_SetPoint := 'False'} : Array[0..10] of "Time_S";
   END_VAR

   VAR_TEMP 
      x : Int;
   END_VAR


BEGIN
	//Получение данных от ЩКД1
	    //контроль связи
	    IF #watchdog_control = #From_SKD1.watchdog THEN
	        #Clock[0].Start := TRUE;
	        IF #Clock[0]."Exit" THEN
	            #Alarm.Link := TRUE; //нет связи с ЩКД1
	        ELSE
	            #Alarm.Link := FALSE;
	        END_IF;
	    ELSE
	        #Clock[0].Start := FALSE;
	    END_IF;
	    
	    //уровни в РВ
	    #LE_1 := INT_TO_REAL(#From_SKD1.LE_1) / 10;
	    #LE_2 := INT_TO_REAL(#From_SKD1.LE_2) / 10;
	    #LE_3 := INT_TO_REAL(#From_SKD1.LE_3) / 10;
	    #LE_4 := INT_TO_REAL(#From_SKD1.LE_4) / 10;
	    
	    //управление насосом
	    IF NOT #To_SKD1.STATE.Local THEN
	        "Pump_DB".CMD.Hand := #From_SKD1.CMD.Hand;
	        "Pump_DB".CMD.Start_M := #From_SKD1.CMD.Start_M;
	        "Pump_DB".SP_M := INT_TO_REAL(#From_SKD1.SP_M) / 10;
	    END_IF;
	    
	    IF #From_SKD1.CMD.Reset THEN
	        "Reset_All" := TRUE;
	    END_IF;
	    
	    //управление
	    "Main_Logick_DB".Start := #From_SKD1.CMD.REQ;
	    "Main_Logick_DB".RM_SP := INT_TO_REAL(#From_SKD1.SP_FE) / 10;
	    
	    IF NOT #From_SKD1.Valves.Local[0] THEN
	        FOR #x := 1 TO 10 BY 1 DO
	            #To_SKD1.Valves.REQ[#x] := #From_SKD1.Valves.Local[#x];
	        END_FOR;
	    END_IF;
	    
	//Передача данных в ЩКД1
	    //контроль связи
	    IF "pulse_1s" THEN
	        #To_SKD1.watchdog := #To_SKD1.watchdog + 1;
	        IF #To_SKD1.watchdog > 10000 THEN
	            #To_SKD1.watchdog := 0;
	        END_IF;
	    END_IF;
	    
	    //состояние установки
	    #To_SKD1.STATE.Ready := "Main_Logick_DB".Ready;
	    #To_SKD1.STATE.Alarm := "Alm_Any";
	    #To_SKD1.STATE.LS := "DIx_1_DB".Level_Norm.Signal;
	    
	    //насос
	    #To_SKD1.res_h := "Pump_DB".OpTime_h;
	    #To_SKD1.Status := "Pump_DB".Status;
	    #To_SKD1.STATE.Lock := "Pump_DB".CMD.Lock;
	    
	    //давление в КП
	    #To_SKD1.PE_1 := REAL_TO_INT("PE_1_DB".Result * 10);
	    #To_SKD1.PE_2 := REAL_TO_INT("PE_2_DB".Result * 10);
	    #To_SKD1.PE_3 := REAL_TO_INT("PE_3_DB".Result * 10);
	    #To_SKD1.PE_4 := REAL_TO_INT("PE_4_DB".Result * 10);
	    
	    //Прочие датчики
	    #To_SKD1.LE := REAL_TO_INT("LE_DB".Result * 10);
	    #To_SKD1.TE := REAL_TO_INT("TE_1_DB".Result * 10);
	    #To_SKD1.FE := REAL_TO_INT("FE_DB".FE[1].Flow * 10);
	    #To_SKD1.C := REAL_TO_INT("C_Pump_DB".Result * 10);
	    
	    //Сброс аварий задвижек
	    IF #To_SKD1.Valves.REQ[0] THEN
	        #Clock[1].Start := TRUE;
	    END_IF;
	    IF #Clock[1]."Exit" THEN
	        #To_SKD1.Valves.REQ[0] := FALSE;
	        #Clock[1].Start := FALSE;
	    END_IF;
	    
	    
	//вызов таймеров на исполнение
	FOR #x := 0 TO 10 BY 1 DO
	    #Clock[#x]();
	END_FOR;
END_FUNCTION_BLOCK

FUNCTION_BLOCK "System"
{ S7_Optimized_Access := 'FALSE' }
VERSION : 0.1
   VAR 
      PE_1_Delta : Real;
      PE_2_Detla : Real;
      PE_1_Min : Real := 0.2;
      PE_2_Min : Real;
   END_VAR


BEGIN
	//Отключение аварий
	IF NOT "Pump_DB".ON THEN
	    "C_Pump_DB".Use.Lim_Low := TRUE;
	    "PE_1_DB".Use.Lim_Low := TRUE;
	    "PE_2_DB".Use.Lim_Low := TRUE;
	ELSE
	    "C_Pump_DB".Use.Lim_Low := FALSE;
	    "PE_1_DB".Use.Lim_Low := FALSE;
	    "PE_2_DB".Use.Lim_Low := FALSE;
	END_IF;
	
	//Снижение расхода при высоком давлении
	IF "PE_1_DB".Alarm.H THEN
	    #PE_1_Delta := "PE_1_DB".SP.HH - "PE_1_DB".Result;
	    IF #PE_1_Delta > 1 THEN
	        #PE_1_Delta := 1.0;
	    END_IF;
	    IF #PE_1_Delta < #PE_1_Min THEN
	        "Pump_DB".CMD.Lock := TRUE;
	        #PE_1_Delta := #PE_1_Min;
	    END_IF;
	    "Pump_DB".coeff := #PE_1_Delta;
	ELSE
	    "Pump_DB".coeff := 1.0;
	END_IF;
	
	//Возобновление работы
	IF "Reset_All" THEN
	    "Pump_DB".CMD.Lock := FALSE;
	END_IF;
	
	//костыль для управления насосами
	IF "Pump_DB".Indirect_BIT.CMD = 0 THEN
	    "Tag_2" := "Pump_DB".CMD_Run;
	END_IF;
END_FUNCTION_BLOCK

FUNCTION_BLOCK "DOx_1"   // FB210, LAD
{ S7_Optimized_Access := 'FALSE' }
VERSION : 0.1
// Start - управляющий сигнал из программы
// Q - выходной сигнал контроллера
// pulse - кратность времени в импульсном режиме
// stored: AutoNumber false, IsIECCheckEnabled false, SetENOAutomatically false, UDAEnableTagReadback false
   VAR
      All_Alarm { S7_SetPoint := 'True'} : "DO_ex";   // Общая авария
      command_2 { S7_SetPoint := 'True'} : "DO_ex";
      command_3 { S7_SetPoint := 'True'} : "DO_ex";
      command_4 { S7_SetPoint := 'True'} : "DO_ex";
      command_5 { S7_SetPoint := 'True'} : "DO_ex";
      command_6 { S7_SetPoint := 'True'} : "DO_ex";
      command_7 { S7_SetPoint := 'True'} : "DO_ex";
      command_8 { S7_SetPoint := 'True'} : "DO_ex";
      command_9 { S7_SetPoint := 'True'} : "DO_ex";
      command_10 { S7_SetPoint := 'True'} : "DO_ex";
      command_11 { S7_SetPoint := 'True'} : "DO_ex";
      command_12 { S7_SetPoint := 'True'} : "DO_ex";
   END_VAR
   VAR DB_SPECIFIC
      Time_DTL { S7_SetPoint := 'True'} : DTL;
   END_VAR
   // All_Alarm.ADDR_Bit := 1;
   VAR_TEMP   // added for the SCL form of the ladder/FBD networks
      _w1 : Bool;
   END_VAR
BEGIN

REGION Network 1
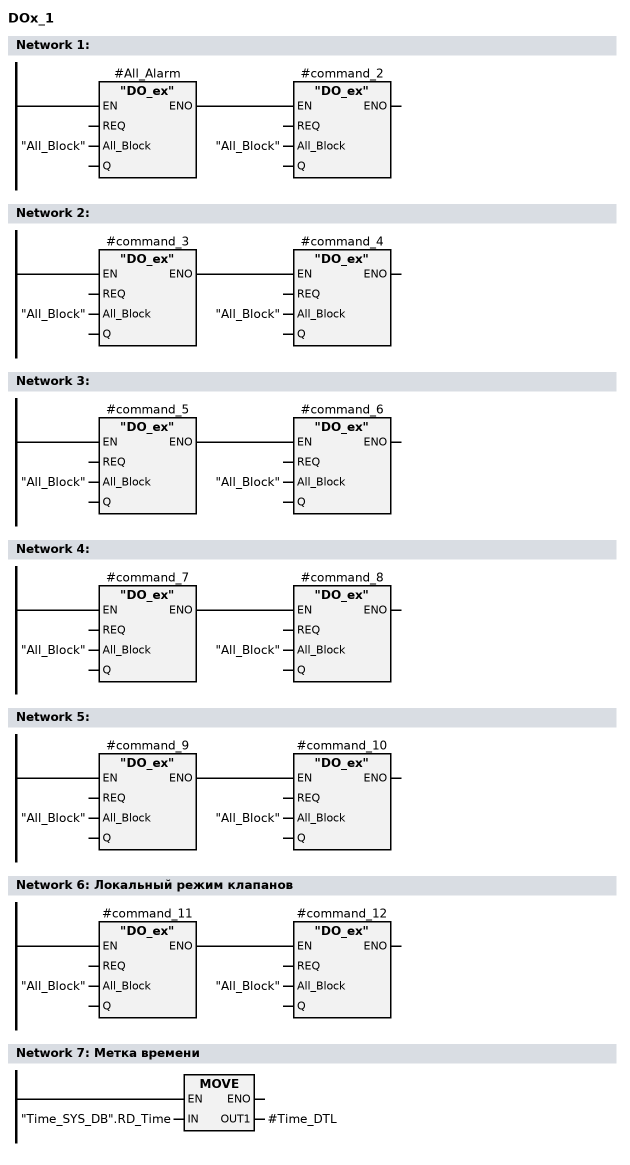
   RUNG wire#powerrail
      #All_Alarm(REQ :=, All_Block := "All_Block", Q :=)
      #command_2(REQ :=, All_Block := "All_Block", Q :=)
   END_RUNG
   // the same network as SCL:
   #All_Alarm(All_Block := "All_Block", ENO => #_w1);   // "DO_ex"
   IF #_w1 THEN
       #command_2(All_Block := "All_Block");   // "DO_ex"
   END_IF;
END_REGION

REGION Network 2
   RUNG wire#powerrail
      #command_3(REQ :=, All_Block := "All_Block", Q :=)
      #command_4(REQ :=, All_Block := "All_Block", Q :=)
   END_RUNG
   // the same network as SCL:
   #command_3(All_Block := "All_Block", ENO => #_w1);   // "DO_ex"
   IF #_w1 THEN
       #command_4(All_Block := "All_Block");   // "DO_ex"
   END_IF;
END_REGION

REGION Network 3
   RUNG wire#powerrail
      #command_5(REQ :=, All_Block := "All_Block", Q :=)
      #command_6(REQ :=, All_Block := "All_Block", Q :=)
   END_RUNG
   // the same network as SCL:
   #command_5(All_Block := "All_Block", ENO => #_w1);   // "DO_ex"
   IF #_w1 THEN
       #command_6(All_Block := "All_Block");   // "DO_ex"
   END_IF;
END_REGION

REGION Network 4
   RUNG wire#powerrail
      #command_7(REQ :=, All_Block := "All_Block", Q :=)
      #command_8(REQ :=, All_Block := "All_Block", Q :=)
   END_RUNG
   // the same network as SCL:
   #command_7(All_Block := "All_Block", ENO => #_w1);   // "DO_ex"
   IF #_w1 THEN
       #command_8(All_Block := "All_Block");   // "DO_ex"
   END_IF;
END_REGION

REGION Network 5
   RUNG wire#powerrail
      #command_9(REQ :=, All_Block := "All_Block", Q :=)
      #command_10(REQ :=, All_Block := "All_Block", Q :=)
   END_RUNG
   // the same network as SCL:
   #command_9(All_Block := "All_Block", ENO => #_w1);   // "DO_ex"
   IF #_w1 THEN
       #command_10(All_Block := "All_Block");   // "DO_ex"
   END_IF;
END_REGION

REGION Network 6: Локальный режим клапанов
   RUNG wire#powerrail
      #command_11(REQ :=, All_Block := "All_Block", Q :=)
      #command_12(REQ :=, All_Block := "All_Block", Q :=)
   END_RUNG
   // the same network as SCL:
   #command_11(All_Block := "All_Block", ENO => #_w1);   // "DO_ex"
   IF #_w1 THEN
       #command_12(All_Block := "All_Block");   // "DO_ex"
   END_IF;
END_REGION

REGION Network 7: Метка времени
   RUNG wire#powerrail
      Move(in := "Time_SYS_DB".RD_Time, out1 => #Time_DTL)
   END_RUNG
   // the same network as SCL:
   #Time_DTL := "Time_SYS_DB".RD_Time;
END_REGION
END_FUNCTION_BLOCK

FUNCTION_BLOCK "DO_ex"   // FB102, LAD
{ S7_Optimized_Access := 'FALSE' }
VERSION : 0.1
// stored: AutoNumber false, IsIECCheckEnabled false, SetENOAutomatically false, UDAEnableTagReadback false
   VAR_INPUT
      REQ : Bool;   // Запрос включения
      All_Block : Bool;
   END_VAR
   VAR_IN_OUT
      Q : Bool;   // Выходной сигнал ПЛК
   END_VAR
   VAR DB_SPECIFIC
      CMD : "CMD";   // Основные команды / Блок команд
      Use : Struct   // Функционал
         Inverse { S7_SetPoint := 'True'} : Bool;   // Инверсия входного сигнала
         Indirect { S7_SetPoint := 'True'} : Bool := true;   // Использование косвенной адресации
         Impulse { S7_SetPoint := 'True'} : Bool;   // Использовать импульсный режим
      END_STRUCT;
      ADDR_Byte { S7_SetPoint := 'True'} : Int;   // Адрес входа на контроллере (Байт)
      ADDR_Bit { S7_SetPoint := 'True'} : Int := 9;   // Адрес входа на контроллере (Бит)
      Mode : Int;
      Status : Int;
   END_VAR
   VAR
      T_Impulse { S7_SetPoint := 'True'} : "Time_S_b";   // Длительность импульса
   END_VAR
   VAR_TEMP
      Start : Bool;
   END_VAR
   VAR_TEMP   // added for the SCL form of the ladder/FBD networks
      _w1 : Bool;
   END_VAR
BEGIN

REGION Network 1: Устройство в ручном режиме
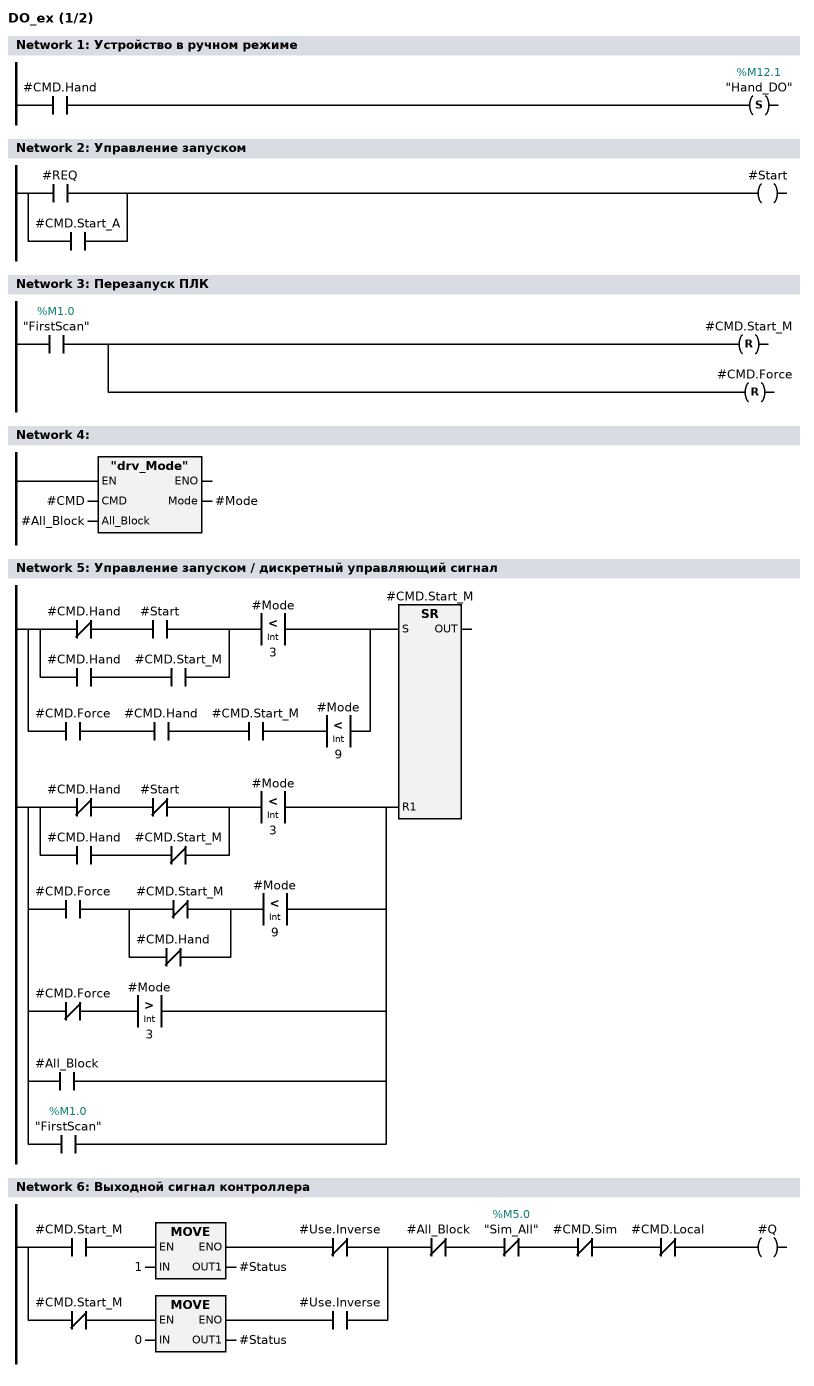
   RUNG wire#powerrail
      Contact( #CMD.Hand )
      S_Coil( "Hand_DO" )
   END_RUNG
   // the same network as SCL:
   IF #CMD.Hand THEN "Hand_DO" := TRUE; END_IF;
END_REGION

REGION Network 2: Управление запуском
   RUNG wire#powerrail
      Contact( #REQ )
      wire#w1
      Coil( #Start )
   END_RUNG
   RUNG wire#powerrail
      Contact( #CMD.Start_A )
   END_RUNG wire#w1
   // the same network as SCL:
   #Start := #REQ OR #CMD.Start_A;
END_REGION

REGION Network 3: Перезапуск ПЛК
   RUNG wire#powerrail
      Contact( "FirstScan" )
      wire#w1
      R_Coil( #CMD.Start_M )
   END_RUNG
   RUNG wire#w1
      R_Coil( #CMD.Force )
   END_RUNG
   // the same network as SCL:
   IF "FirstScan" THEN
       #CMD.Start_M := FALSE;
       #CMD.Force := FALSE;
   END_IF;
END_REGION

REGION Network 4
   RUNG wire#powerrail
      "drv_Mode"(CMD := #CMD, All_Block := #All_Block, Mode => #Mode)
   END_RUNG
   // the same network as SCL:
   "drv_Mode"(CMD := #CMD, All_Block := #All_Block, Mode => #Mode);
END_REGION

REGION Network 5: Управление запуском / дискретный управляющий сигнал
   RUNG wire#powerrail
      I_Contact( #CMD.Hand )
      Contact( #Start )
      wire#w1
      { S7_Templates := "SrcType := Int" } LT_Contact(in1 := #Mode, in2 := 3)
      wire#w2
      S_SR(operand := #CMD.Start_M, r1 := wire#w6)
   END_RUNG
   RUNG wire#powerrail
      Contact( #CMD.Hand )
      Contact( #CMD.Start_M )
   END_RUNG wire#w1
   RUNG wire#powerrail
      Contact( #CMD.Force )
      Contact( #CMD.Hand )
      Contact( #CMD.Start_M )
      { S7_Templates := "SrcType := Int" } LT_Contact(in1 := #Mode, in2 := 9)
   END_RUNG wire#w2
   RUNG wire#powerrail
      I_Contact( #CMD.Hand )
      I_Contact( #Start )
      wire#w3
      { S7_Templates := "SrcType := Int" } LT_Contact(in1 := #Mode, in2 := 3)
   END_RUNG wire#w6
   RUNG wire#powerrail
      Contact( #CMD.Hand )
      I_Contact( #CMD.Start_M )
   END_RUNG wire#w3
   RUNG wire#powerrail
      Contact( #CMD.Force )
      wire#w4
      I_Contact( #CMD.Start_M )
      wire#w5
      { S7_Templates := "SrcType := Int" } LT_Contact(in1 := #Mode, in2 := 9)
   END_RUNG wire#w6
   RUNG wire#w4
      I_Contact( #CMD.Hand )
   END_RUNG wire#w5
   RUNG wire#powerrail
      I_Contact( #CMD.Force )
      { S7_Templates := "SrcType := Int" } GT_Contact(in1 := #Mode, in2 := 3)
   END_RUNG wire#w6
   RUNG wire#powerrail
      Contact( #All_Block )
   END_RUNG wire#w6
   RUNG wire#powerrail
      Contact( "FirstScan" )
   END_RUNG wire#w6
   // the same network as SCL:
   #_w1 := (((NOT #CMD.Hand AND NOT #Start) OR (#CMD.Hand AND NOT #CMD.Start_M)) AND (#Mode < 3)) OR (#CMD.Force AND (NOT #CMD.Start_M OR NOT #CMD.Hand) AND (#Mode < 9)) OR (NOT #CMD.Force AND (#Mode > 3)) OR #All_Block OR "FirstScan";
   IF (((NOT #CMD.Hand AND #Start) OR (#CMD.Hand AND #CMD.Start_M)) AND (#Mode < 3)) OR (#CMD.Force AND #CMD.Hand AND #CMD.Start_M AND (#Mode < 9)) THEN
       #CMD.Start_M := TRUE;   // SR flip-flop
   END_IF;
   IF #_w1 THEN #CMD.Start_M := FALSE; END_IF;
END_REGION

